KUKA KRL program: EPS_2_251825_SA33_A_20260116064116.src

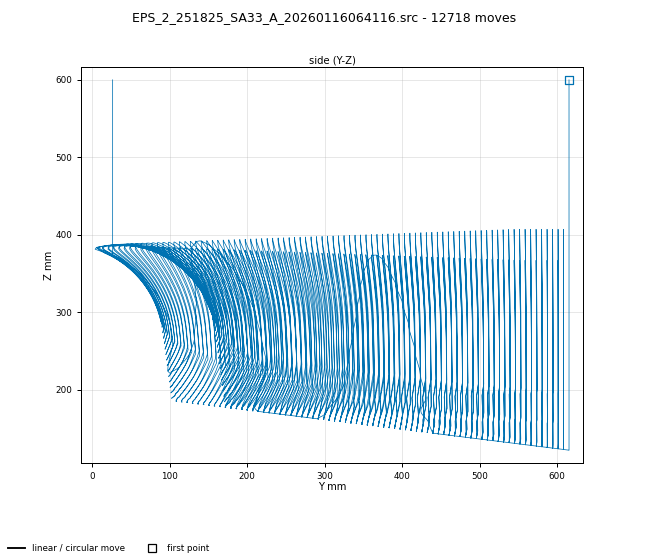
[picture p0: tool path of EPS_2_251825_SA33_A_20260116064116.src, 12718 of 12720 moves have a stored position in this frame; points joined in program order, loops and branches not executed]
&ACCESS RVP
&REL 4
&COMMENT QRS 19112012
&PARAM EDITMASK = *
DEF PART()
EXT BAS (BAS_COMMAND :IN,REAL :IN )
INT I
BAS (#INITMOV,0 )

;KUKA QRS Post kuka4.cps  Date:22-06-2017 !

File_ID=2980

QRS_PRE_INIT()

;Init var - Until changes are made in qrs_pre_init
Outlet_Square_prg=0
Inlet_1_Square_prg=0
Inlet_2_Square_prg=0
Inlet_3_Square_prg=0
Inlet_4_Square_prg=0
Inlet_5_Square_prg=0

Outlet_1={X 0.000, Y 546.330, Z 306.500, B 0.000, E1 0.000 }
Inlet_1={X 0.000, Y 549.180, Z 266.500, B 0.000, E1 202.000 }
Outlet_1_type=201
Inlet_1_type=201
;QRS#1=Sidecore dimensions
;QRS#2=200-8" PVC SDR 35
;QRS#3=200-8" PVC SDR 35
;QRS#4=
;QRS#5=
;QRS#6=
;QRS#7=
;QRS#8=
;QRS#9=12-08 PSX
;QRS#10=12-08 PSX
;QRS#11=
;QRS#12=
;QRS#13=
;QRS#14=
;QRS#15=
;QRS#16=1220x127x686 2,25'
;QRS#17=EPS Height
;QRS#18=407
;QRS#19=*
;QRS#20= UPDATED VERSION 22-06-2017
;QRS#21=*
Outlet_Square=0100
Inlet_1_Square=0100
Inlet_2_Square=0
Inlet_3_Square=0
Inlet_4_Square=0
Inlet_5_Square=0
Mill_Square=1
Outlet_Square_Prg=204
Inlet_1_Square_prg=204

QRS_INIT()

$ADVANCE=5

; T1
PTP {E1 173.647,E2 173.647}
PTP {X 0,Y 615.463,A -85,B 0,C 180,E1 173.647,E2 173.647,E3 0,E4 0,E5 0,E6 0}
QRS_SPEED_INIT()
LIN {X 0,Y 615.463,Z 600,A -85,B 0,C 180,E1 173.647,E2 173.647,E3 0,E4 0,E5 0,E6 0} C_VEL
LIN {X 0,Y 615.463,Z 131.877,A -85,B 0,C 180,E1 173.647,E2 173.647} C_VEL
LIN {X 0,Y 615.463,Z 123.698,A -85,B 0,C 180,E1 173.647,E2 173.647} C_VEL
LIN {X 0,Y 615.445,Z 121.698,A -85,B 0,C 180,E1 173.461,E2 173.461} C_VEL
LIN {X 0,Y 615.439,Z 121.698,A -85,B 0,C 180,E1 171.463,E2 171.463} C_VEL
LIN {X 0,Y 615.428,Z 121.696,A -85,B 0,C 180,E1 169.143,E2 169.143} C_VEL
LIN {X 0,Y 615.442,Z 121.695,A -85,B 0,C 180,E1 166.798,E2 166.798} C_VEL
LIN {X 0,Y 615.481,Z 121.702,A -85,B 0,C 180,E1 164.095,E2 164.095} C_VEL
LIN {X 0,Y 615.427,Z 121.697,A -85,B 0,C 180,E1 161.353,E2 161.353} C_VEL
LIN {X 0,Y 615.486,Z 121.694,A -85,B 0,C 180,E1 158.569,E2 158.569} C_VEL
LIN {X 0,Y 615.433,Z 121.698,A -85,B 0,C 180,E1 155.726,E2 155.726} C_VEL
LIN {X 0,Y 615.425,Z 121.697,A -85,B 0,C 180,E1 153.554,E2 153.554} C_VEL
LIN {X 0,Y 615.493,Z 121.698,A -85,B 0,C 180,E1 150.595,E2 150.595} C_VEL
LIN {X 0,Y 615.468,Z 121.699,A -85,B 0,C 180,E1 148.314,E2 148.314} C_VEL
LIN {X 0,Y 615.433,Z 121.698,A -85,B 0,C 180,E1 145.975,E2 145.975} C_VEL
LIN {X 0,Y 615.427,Z 121.697,A -85,B 0,C 180,E1 143.572,E2 143.572} C_VEL
LIN {X 0,Y 615.49,Z 121.695,A -85,B 0,C 180,E1 140.938,E2 140.938} C_VEL
LIN {X 0,Y 615.465,Z 121.699,A -85,B 0,C 180,E1 138.525,E2 138.525} C_VEL
LIN {X 0,Y 615.424,Z 121.698,A -85,B 0,C 180,E1 136.009,E2 136.009} C_VEL
LIN {X 0,Y 615.423,Z 121.698,A -85,B 0,C 180,E1 133.992,E2 133.992} C_VEL
LIN {X 0,Y 615.448,Z 121.696,A -85,B 0,C 180,E1 131.478,E2 131.478} C_VEL
LIN {X 0,Y 615.485,Z 121.7,A -85,B 0,C 180,E1 128.905,E2 128.905} C_VEL
LIN {X 0,Y 615.43,Z 121.698,A -85,B 0,C 180,E1 126.429,E2 126.429} C_VEL
LIN {X 0,Y 615.422,Z 121.698,A -85,B 0,C 180,E1 124.026,E2 124.026} C_VEL
LIN {X 0,Y 615.445,Z 121.697,A -85,B 0,C 180,E1 121.688,E2 121.688} C_VEL
LIN {X 0,Y 615.479,Z 121.698,A -85,B 0,C 180,E1 119.407,E2 119.407} C_VEL
LIN {X 0,Y 615.421,Z 121.698,A -85,B 0,C 180,E1 116.448,E2 116.448} C_VEL
LIN {X 0,Y 615.436,Z 121.697,A -85,B 0,C 180,E1 113.999,E2 113.999} C_VEL
LIN {X 0,Y 615.498,Z 121.7,A -85,B 0,C 180,E1 111.432,E2 111.432} C_VEL
LIN {X 0,Y 615.419,Z 121.698,A -85,B 0,C 180,E1 108.588,E2 108.588} C_VEL
LIN {X 0,Y 615.462,Z 121.697,A -85,B 0,C 180,E1 105.906,E2 105.906} C_VEL
LIN {X 0,Y 615.444,Z 121.699,A -85,B 0,C 180,E1 103.202,E2 103.202} C_VEL
LIN {X 0,Y 615.417,Z 121.699,A -85,B 0,C 180,E1 100.858,E2 100.858} C_VEL
LIN {X 0,Y 615.423,Z 121.698,A -85,B 0,C 180,E1 98.538,E2 98.538} C_VEL
LIN {X 0,Y 615.496,Z 121.697,A -85,B 0,C 180,E1 95.899,E2 95.899} C_VEL
LIN {X 0,Y 615.429,Z 121.699,A -85,B 0,C 180,E1 93.273,E2 93.273} C_VEL
LIN {X 0,Y 615.429,Z 121.699,A -85,B 0,C 180,E1 91.309,E2 91.309} C_VEL
LIN {X 0,Y 615.427,Z 121.699,A -85,B 0,C 180,E1 89.346,E2 89.346} C_VEL
LIN {X 0,Y 615.427,Z 121.699,A -85,B 0,C 180,E1 87.382,E2 87.382} C_VEL
LIN {X 0,Y 615.434,Z 121.811,A -85,B 0,C 180,E1 86.604,E2 86.604} C_VEL
LIN {X 0,Y 615.454,Z 138.456,A -85,B 0,C 180,E1 83.781,E2 83.781} C_VEL
LIN {X 0,Y 615.439,Z 154.279,A -85,B 0,C 180,E1 81.132,E2 81.132} C_VEL
LIN {X 0,Y 615.46,Z 156.135,A -85,B 0,C 180,E1 80.822,E2 80.822} C_VEL
LIN {X 0,Y 615.446,Z 263.403,A -85,B 0,C 180,E1 79.535,E2 79.535} C_VEL
LIN {X 0,Y 615.449,Z 276.074,A -85,B 0,C 180,E1 79.254,E2 79.254} C_VEL
LIN {X 0,Y 615.477,Z 288.507,A -85,B 0,C 180,E1 78.846,E2 78.846} C_VEL
LIN {X 0,Y 615.497,Z 300.645,A -85,B 0,C 180,E1 78.307,E2 78.307} C_VEL
LIN {X 0,Y 615.483,Z 312.21,A -85,B 0,C 180,E1 77.637,E2 77.637} C_VEL
LIN {X 0,Y 615.498,Z 322.624,A -85,B 0,C 180,E1 76.883,E2 76.883} C_VEL
LIN {X 0,Y 615.497,Z 331.842,A -85,B 0,C 180,E1 76.06,E2 76.06} C_VEL
LIN {X 0,Y 615.496,Z 340.437,A -85,B 0,C 180,E1 75.113,E2 75.113} C_VEL
LIN {X 0,Y 615.497,Z 347.906,A -85,B 0,C 180,E1 74.095,E2 74.095} C_VEL
LIN {X 0,Y 615.496,Z 353.873,A -85,B 0,C 180,E1 73.072,E2 73.072} C_VEL
LIN {X 0,Y 615.498,Z 358.543,A -85,B 0,C 180,E1 72.043,E2 72.043} C_VEL
LIN {X 0,Y 615.494,Z 362.068,A -85,B 0,C 180,E1 71.009,E2 71.009} C_VEL
LIN {X 0,Y 615.495,Z 364.527,A -85,B 0,C 180,E1 69.967,E2 69.967} C_VEL
LIN {X 0,Y 615.497,Z 365.572,A -85,B 0,C 180,E1 69.27,E2 69.27} C_VEL
LIN {X 0,Y 615.498,Z 366.202,A -85,B 0,C 180,E1 68.569,E2 68.569} C_VEL
LIN {X 0,Y 615.497,Z 366.321,A -85,B 0,C 180,E1 67.65,E2 67.65} C_VEL
LIN {X 0,Y 615.496,Z 365.342,A -85,B 0,C 180,E1 66.444,E2 66.444} C_VEL
LIN {X 0,Y 615.494,Z 364.093,A -85,B 0,C 180,E1 65.728,E2 65.728} C_VEL
LIN {X 0,Y 615.495,Z 362.354,A -85,B 0,C 180,E1 65.009,E2 65.009} C_VEL
LIN {X 0,Y 615.496,Z 358.747,A -85,B 0,C 180,E1 63.921,E2 63.921} C_VEL
LIN {X 0,Y 615.494,Z 353.798,A -85,B 0,C 180,E1 62.823,E2 62.823} C_VEL
LIN {X 0,Y 615.496,Z 347.915,A -85,B 0,C 180,E1 61.816,E2 61.816} C_VEL
LIN {X 0,Y 615.496,Z 340.312,A -85,B 0,C 180,E1 60.782,E2 60.782} C_VEL
LIN {X 0,Y 615.496,Z 331.75,A -85,B 0,C 180,E1 59.84,E2 59.84} C_VEL
LIN {X 0,Y 615.497,Z 322.228,A -85,B 0,C 180,E1 58.996,E2 58.996} C_VEL
LIN {X 0,Y 615.471,Z 311.616,A -85,B 0,C 180,E1 58.234,E2 58.234} C_VEL
LIN {X 0,Y 615.467,Z 300.715,A -85,B 0,C 180,E1 57.606,E2 57.606} C_VEL
LIN {X 0,Y 615.494,Z 288.315,A -85,B 0,C 180,E1 57.057,E2 57.057} C_VEL
LIN {X 0,Y 615.49,Z 275.924,A -85,B 0,C 180,E1 56.653,E2 56.653} C_VEL
LIN {X 0,Y 615.467,Z 263.343,A -85,B 0,C 180,E1 56.375,E2 56.375} C_VEL
LIN {X 0,Y 615.49,Z 156.109,A -85,B 0,C 180,E1 55.085,E2 55.085} C_VEL
LIN {X 0,Y 615.471,Z 139.904,A -85,B 0,C 180,E1 52.373,E2 52.373} C_VEL
LIN {X 0,Y 615.484,Z 123.817,A -85,B 0,C 180,E1 49.651,E2 49.651} C_VEL
LIN {X 0,Y 615.48,Z 121.688,A -85,B 0,C 180,E1 49.271,E2 49.271} C_VEL
LIN {X 0,Y 615.486,Z 121.684,A -85,B 0,C 180,E1 46.755,E2 46.755} C_VEL
LIN {X 0,Y 615.488,Z 121.7,A -85,B 0,C 180,E1 43.997,E2 43.997} C_VEL
LIN {X 0,Y 615.487,Z 121.683,A -85,B 0,C 180,E1 41.094,E2 41.094} C_VEL
LIN {X 0,Y 615.487,Z 121.686,A -85,B 0,C 180,E1 38.903,E2 38.903} C_VEL
LIN {X 0,Y 615.487,Z 121.7,A -85,B 0,C 180,E1 36.424,E2 36.424} C_VEL
LIN {X 0,Y 615.478,Z 121.685,A -85,B 0,C 180,E1 33.533,E2 33.533} C_VEL
LIN {X 0,Y 615.484,Z 121.691,A -85,B 0,C 180,E1 30.919,E2 30.919} C_VEL
LIN {X 0,Y 615.484,Z 121.698,A -85,B 0,C 180,E1 28.449,E2 28.449} C_VEL
LIN {X 0,Y 615.483,Z 121.685,A -85,B 0,C 180,E1 25.567,E2 25.567} C_VEL
LIN {X 0,Y 615.49,Z 121.7,A -85,B 0,C 180,E1 22.844,E2 22.844} C_VEL
LIN {X 0,Y 615.472,Z 121.696,A -85,B 0,C 180,E1 20.553,E2 20.553} C_VEL
LIN {X 0,Y 615.468,Z 121.687,A -85,B 0,C 180,E1 17.957,E2 17.957} C_VEL
LIN {X 0,Y 615.493,Z 121.695,A -85,B 0,C 180,E1 15.225,E2 15.225} C_VEL
LIN {X 0,Y 615.457,Z 121.693,A -85,B 0,C 180,E1 12.53,E2 12.53} C_VEL
LIN {X 0,Y 615.491,Z 121.685,A -85,B 0,C 180,E1 9.862,E2 9.862} C_VEL
LIN {X 0,Y 615.48,Z 121.701,A -85,B 0,C 180,E1 7.215,E2 7.215} C_VEL
LIN {X 0,Y 615.451,Z 121.692,A -85,B 0,C 180,E1 4.584,E2 4.584} C_VEL
LIN {X 0,Y 615.5,Z 121.686,A -85,B 0,C 180,E1 1.963,E2 1.963} C_VEL
LIN {X 0,Y 615.472,Z 121.698,A -85,B 0,C 180,E1 -0.655,E2 -0.655} C_VEL
LIN {X 0,Y 615.469,Z 121.698,A -85,B 0,C 180,E1 -2.618,E2 -2.618} C_VEL
LIN {X 0,Y 615.443,Z 121.693,A -85,B 0,C 180,E1 -5.242,E2 -5.242} C_VEL
LIN {X 0,Y 615.489,Z 121.693,A -85,B 0,C 180,E1 -7.876,E2 -7.876} C_VEL
LIN {X 0,Y 615.452,Z 121.697,A -85,B 0,C 180,E1 -10.528,E2 -10.528} C_VEL
LIN {X 0,Y 615.446,Z 121.697,A -85,B 0,C 180,E1 -12.531,E2 -12.531} C_VEL
LIN {X 0,Y 615.437,Z 121.698,A -85,B 0,C 180,E1 -14.551,E2 -14.551} C_VEL
LIN {X 0,Y 615.435,Z 121.697,A -85,B 0,C 180,E1 -16.589,E2 -16.589} C_VEL
LIN {X 0,Y 615.431,Z 121.696,A -85,B 0,C 180,E1 -18.648,E2 -18.648} C_VEL
LIN {X 0,Y 615.487,Z 121.694,A -85,B 0,C 180,E1 -21.432,E2 -21.432} C_VEL
LIN {X 0,Y 615.432,Z 121.698,A -85,B 0,C 180,E1 -24.275,E2 -24.275} C_VEL
LIN {X 0,Y 615.42,Z 121.699,A -85,B 0,C 180,E1 -26.448,E2 -26.448} C_VEL
LIN {X 0,Y 615.491,Z 121.701,A -85,B 0,C 180,E1 -29.407,E2 -29.407} C_VEL
LIN {X 0,Y 615.455,Z 121.7,A -85,B 0,C 180,E1 -31.688,E2 -31.688} C_VEL
LIN {X 0,Y 615.421,Z 121.7,A -85,B 0,C 180,E1 -34.027,E2 -34.027} C_VEL
LIN {X 0,Y 615.463,Z 121.7,A -85,B 0,C 180,E1 -36.933,E2 -36.933} C_VEL
LIN {X 0,Y 615.422,Z 121.7,A -85,B 0,C 180,E1 -39.756,E2 -39.756} C_VEL
LIN {X 0,Y 615.416,Z 121.699,A -85,B 0,C 180,E1 -42.073,E2 -42.073} C_VEL
LIN {X 0,Y 615.421,Z 121.699,A -85,B 0,C 180,E1 -44.156,E2 -44.156} C_VEL
LIN {X 0,Y 615.484,Z 121.7,A -85,B 0,C 180,E1 -46.755,E2 -46.755} C_VEL
LIN {X 0,Y 615.441,Z 121.697,A -85,B 0,C 180,E1 -49.39,E2 -49.39} C_VEL
LIN {X 0,Y 615.428,Z 121.698,A -85,B 0,C 180,E1 -51.927,E2 -51.927} C_VEL
LIN {X 0,Y 615.47,Z 121.699,A -85,B 0,C 180,E1 -54.383,E2 -54.383} C_VEL
LIN {X 0,Y 615.486,Z 121.695,A -85,B 0,C 180,E1 -56.764,E2 -56.764} C_VEL
LIN {X 0,Y 615.453,Z 121.693,A -85,B 0,C 180,E1 -59.078,E2 -59.078} C_VEL
LIN {X 0,Y 615.435,Z 121.696,A -85,B 0,C 180,E1 -61.559,E2 -61.559} C_VEL
LIN {X 0,Y 615.494,Z 121.695,A -85,B 0,C 180,E1 -64.431,E2 -64.431} C_VEL
LIN {X 0,Y 615.442,Z 121.693,A -85,B 0,C 180,E1 -67.154,E2 -67.154} C_VEL
LIN {X 0,Y 615.441,Z 121.788,A -85,B 0,C 180,E1 -67.44,E2 -67.44} C_VEL
LIN {X 0,Y 615.477,Z 140.398,A -85,B 0,C 180,E1 -69.967,E2 -69.967} C_VEL
LIN {X 0,Y 615.47,Z 161.077,A -85,B 0,C 180,E1 -72.729,E2 -72.729} C_VEL
LIN {X 0,Y 615.472,Z 181.733,A -85,B 0,C 180,E1 -75.451,E2 -75.451} C_VEL
LIN {X 0,Y 615.454,Z 194.471,A -85,B 0,C 180,E1 -77.113,E2 -77.113} C_VEL
LIN {X 0,Y 615.488,Z 302.833,A -85,B 0,C 180,E1 -78.411,E2 -78.411} C_VEL
LIN {X 0,Y 615.477,Z 315.348,A -85,B 0,C 180,E1 -78.682,E2 -78.682} C_VEL
LIN {X 0,Y 615.488,Z 328.62,A -85,B 0,C 180,E1 -79.113,E2 -79.113} C_VEL
LIN {X 0,Y 615.477,Z 340.48,A -85,B 0,C 180,E1 -79.639,E2 -79.639} C_VEL
LIN {X 0,Y 615.494,Z 351.995,A -85,B 0,C 180,E1 -80.304,E2 -80.304} C_VEL
LIN {X 0,Y 615.499,Z 362.342,A -85,B 0,C 180,E1 -81.05,E2 -81.05} C_VEL
LIN {X 0,Y 615.497,Z 370.813,A -85,B 0,C 180,E1 -81.794,E2 -81.794} C_VEL
LIN {X 0,Y 615.498,Z 378.607,A -85,B 0,C 180,E1 -82.62,E2 -82.62} C_VEL
LIN {X 0,Y 615.496,Z 386.204,A -85,B 0,C 180,E1 -83.608,E2 -83.608} C_VEL
LIN {X 0,Y 615.498,Z 393.205,A -85,B 0,C 180,E1 -84.759,E2 -84.759} C_VEL
LIN {X 0,Y 615.494,Z 397.852,A -85,B 0,C 180,E1 -85.744,E2 -85.744} C_VEL
LIN {X 0,Y 615.494,Z 401.399,A -85,B 0,C 180,E1 -86.727,E2 -86.727} C_VEL
LIN {X 0,Y 615.497,Z 403.233,A -85,B 0,C 180,E1 -87.382,E2 -87.382} C_VEL
LIN {X 0,Y 615.5,Z 404.608,A -85,B 0,C 180,E1 -88.037,E2 -88.037} C_VEL
LIN {X 0,Y 615.496,Z 406.174,A -85,B 0,C 180,E1 -89.346,E2 -89.346} C_VEL
LIN {X 0,Y 615.494,Z 406.389,A -85,B 0,C 180,E1 -90,E2 -90} C_VEL
LIN {X 0,Y 615.495,Z 405.58,A -85,B 0,C 180,E1 -91.309,E2 -91.309} C_VEL
LIN {X 0,Y 615.5,Z 404.607,A -85,B 0,C 180,E1 -91.963,E2 -91.963} C_VEL
LIN {X 0,Y 615.497,Z 403.233,A -85,B 0,C 180,E1 -92.618,E2 -92.618} C_VEL
LIN {X 0,Y 615.496,Z 400.349,A -85,B 0,C 180,E1 -93.601,E2 -93.601} C_VEL
LIN {X 0,Y 615.498,Z 396.441,A -85,B 0,C 180,E1 -94.585,E2 -94.585} C_VEL
LIN {X 0,Y 615.499,Z 391.404,A -85,B 0,C 180,E1 -95.57,E2 -95.57} C_VEL
LIN {X 0,Y 615.497,Z 384.87,A -85,B 0,C 180,E1 -96.583,E2 -96.583} C_VEL
LIN {X 0,Y 615.497,Z 377.131,A -85,B 0,C 180,E1 -97.546,E2 -97.546} C_VEL
LIN {X 0,Y 615.498,Z 369.043,A -85,B 0,C 180,E1 -98.371,E2 -98.371} C_VEL
LIN {X 0,Y 615.499,Z 359.165,A -85,B 0,C 180,E1 -99.199,E2 -99.199} C_VEL
LIN {X 0,Y 615.488,Z 347.978,A -85,B 0,C 180,E1 -99.945,E2 -99.945} C_VEL
LIN {X 0,Y 615.482,Z 337.019,A -85,B 0,C 180,E1 -100.527,E2 -100.527} C_VEL
LIN {X 0,Y 615.48,Z 324.488,A -85,B 0,C 180,E1 -101.04,E2 -101.04} C_VEL
LIN {X 0,Y 615.479,Z 312.057,A -85,B 0,C 180,E1 -101.402,E2 -101.402} C_VEL
LIN {X 0,Y 615.493,Z 298.449,A -85,B 0,C 180,E1 -101.652,E2 -101.652} C_VEL
LIN {X 0,Y 615.454,Z 194.469,A -85,B 0,C 180,E1 -102.887,E2 -102.887} C_VEL
LIN {X 0,Y 615.496,Z 172.694,A -85,B 0,C 180,E1 -105.735,E2 -105.735} C_VEL
LIN {X 0,Y 615.455,Z 152.319,A -85,B 0,C 180,E1 -108.436,E2 -108.436} C_VEL
LIN {X 0,Y 615.475,Z 132.635,A -85,B 0,C 180,E1 -111.082,E2 -111.082} C_VEL
LIN {X 0,Y 615.44,Z 121.695,A -85,B 0,C 180,E1 -112.592,E2 -112.592} C_VEL
LIN {X 0,Y 615.452,Z 121.692,A -85,B 0,C 180,E1 -114.994,E2 -114.994} C_VEL
LIN {X 0,Y 615.475,Z 121.699,A -85,B 0,C 180,E1 -117.916,E2 -117.916} C_VEL
LIN {X 0,Y 615.449,Z 121.697,A -85,B 0,C 180,E1 -120.163,E2 -120.163} C_VEL
LIN {X 0,Y 615.438,Z 121.694,A -85,B 0,C 180,E1 -122.461,E2 -122.461} C_VEL
LIN {X 0,Y 615.454,Z 121.692,A -85,B 0,C 180,E1 -124.818,E2 -124.818} C_VEL
LIN {X 0,Y 615.497,Z 121.692,A -85,B 0,C 180,E1 -127.242,E2 -127.242} C_VEL
LIN {X 0,Y 615.462,Z 121.698,A -85,B 0,C 180,E1 -129.753,E2 -129.753} C_VEL
LIN {X 0,Y 615.439,Z 121.694,A -85,B 0,C 180,E1 -132.358,E2 -132.358} C_VEL
LIN {X 0,Y 615.497,Z 121.692,A -85,B 0,C 180,E1 -135.068,E2 -135.068} C_VEL
LIN {X 0,Y 615.454,Z 121.698,A -85,B 0,C 180,E1 -137.644,E2 -137.644} C_VEL
LIN {X 0,Y 615.438,Z 121.694,A -85,B 0,C 180,E1 -140.246,E2 -140.246} C_VEL
LIN {X 0,Y 615.488,Z 121.701,A -85,B 0,C 180,E1 -143.064,E2 -143.064} C_VEL
LIN {X 0,Y 615.435,Z 121.695,A -85,B 0,C 180,E1 -145.974,E2 -145.974} C_VEL
LIN {X 0,Y 615.485,Z 121.701,A -85,B 0,C 180,E1 -148.915,E2 -148.915} C_VEL
LIN {X 0,Y 615.438,Z 121.696,A -85,B 0,C 180,E1 -151.559,E2 -151.559} C_VEL
LIN {X 0,Y 615.437,Z 121.696,A -85,B 0,C 180,E1 -153.553,E2 -153.553} C_VEL
LIN {X 0,Y 615.444,Z 121.694,A -85,B 0,C 180,E1 -156.002,E2 -156.002} C_VEL
LIN {X 0,Y 615.498,Z 121.694,A -85,B 0,C 180,E1 -158.568,E2 -158.568} C_VEL
LIN {X 0,Y 615.434,Z 121.696,A -85,B 0,C 180,E1 -161.412,E2 -161.412} C_VEL
LIN {X 0,Y 615.433,Z 121.695,A -85,B 0,C 180,E1 -163.588,E2 -163.588} C_VEL
LIN {X 0,Y 615.475,Z 121.692,A -85,B 0,C 180,E1 -166.125,E2 -166.125} C_VEL
LIN {X 0,Y 615.46,Z 121.699,A -85,B 0,C 180,E1 -168.806,E2 -168.806} C_VEL
LIN {X 0,Y 615.456,Z 121.698,A -85,B 0,C 180,E1 -170.8,E2 -170.8} C_VEL
LIN {X 0,Y 615.453,Z 121.698,A -85,B 0,C 180,E1 -172.783,E2 -172.783} C_VEL
LIN {X 0,Y 615.451,Z 121.698,A -85,B 0,C 180,E1 -174.758,E2 -174.758} C_VEL
LIN {X 0,Y 615.45,Z 121.698,A -85,B 0,C 180,E1 -176.726,E2 -176.726} C_VEL
LIN {X 0,Y 615.449,Z 121.698,A -85,B 0,C 180,E1 -178.691,E2 -178.691} C_VEL
LIN {X 0,Y 615.447,Z 121.698,A -85,B 0,C 180,E1 -180.654,E2 -180.654} C_VEL
LIN {X 0,Y 615.447,Z 121.698,A -85,B 0,C 180,E1 -182.617,E2 -182.617} C_VEL
LIN {X 0,Y 615.445,Z 121.698,A -85,B 0,C 180,E1 -184.584,E2 -184.584} C_VEL
LIN {X 0,Y 615.445,Z 121.698,A -85,B 0,C 180,E1 -186.539,E2 -186.539} C_VEL
LIN {X 0,Y 614.76,Z 121.842,A -85,B 0,C 180,E1 -187.085,E2 -187.085} C_VEL
LIN {X 0,Y 611.917,Z 122.266,A -85,B 0,C 180,E1 -187.972,E2 -187.972} C_VEL
LIN {X 0,Y 609.532,Z 122.568,A -85,B 0,C 180,E1 -188.684,E2 -188.684} C_VEL
LIN {X 0,Y 608.513,Z 122.682,A -85,B 0,C 180,E1 -189.234,E2 -189.234} C_VEL
LIN {X 0,Y 608.432,Z 122.692,A -85,B 0,C 180,E1 -189.42,E2 -189.42} C_VEL
LIN {X 0,Y 608.455,Z 122.697,A -85,B 0,C 180,E1 -191.999,E2 -191.999} C_VEL
LIN {X 0,Y 608.4,Z 122.694,A -85,B 0,C 180,E1 -194.722,E2 -194.722} C_VEL
LIN {X 0,Y 608.411,Z 122.693,A -85,B 0,C 180,E1 -196.785,E2 -196.785} C_VEL
LIN {X 0,Y 608.434,Z 122.697,A -85,B 0,C 180,E1 -199.571,E2 -199.571} C_VEL
LIN {X 0,Y 608.416,Z 122.693,A -85,B 0,C 180,E1 -202.407,E2 -202.407} C_VEL
LIN {X 0,Y 608.414,Z 122.692,A -85,B 0,C 180,E1 -204.572,E2 -204.572} C_VEL
LIN {X 0,Y 608.461,Z 122.691,A -85,B 0,C 180,E1 -207.203,E2 -207.203} C_VEL
LIN {X 0,Y 608.419,Z 122.695,A -85,B 0,C 180,E1 -209.963,E2 -209.963} C_VEL
LIN {X 0,Y 608.412,Z 122.693,A -85,B 0,C 180,E1 -212.514,E2 -212.514} C_VEL
LIN {X 0,Y 608.416,Z 122.695,A -85,B 0,C 180,E1 -214.9,E2 -214.9} C_VEL
LIN {X 0,Y 608.436,Z 122.693,A -85,B 0,C 180,E1 -217.748,E2 -217.748} C_VEL
LIN {X 0,Y 608.399,Z 122.694,A -85,B 0,C 180,E1 -220.323,E2 -220.323} C_VEL
LIN {X 0,Y 608.444,Z 122.695,A -85,B 0,C 180,E1 -222.96,E2 -222.96} C_VEL
LIN {X 0,Y 608.409,Z 122.695,A -85,B 0,C 180,E1 -225.74,E2 -225.74} C_VEL
LIN {X 0,Y 608.408,Z 122.693,A -85,B 0,C 180,E1 -227.934,E2 -227.934} C_VEL
LIN {X 0,Y 608.435,Z 122.695,A -85,B 0,C 180,E1 -230.705,E2 -230.705} C_VEL
LIN {X 0,Y 608.45,Z 122.696,A -85,B 0,C 180,E1 -233.084,E2 -233.084} C_VEL
LIN {X 0,Y 608.425,Z 122.692,A -85,B 0,C 180,E1 -235.527,E2 -235.527} C_VEL
LIN {X 0,Y 608.415,Z 122.692,A -85,B 0,C 180,E1 -237.902,E2 -237.902} C_VEL
LIN {X 0,Y 608.428,Z 122.693,A -85,B 0,C 180,E1 -240.218,E2 -240.218} C_VEL
LIN {X 0,Y 608.467,Z 122.695,A -85,B 0,C 180,E1 -242.793,E2 -242.793} C_VEL
LIN {X 0,Y 608.409,Z 122.693,A -85,B 0,C 180,E1 -245.427,E2 -245.427} C_VEL
LIN {X 0,Y 608.454,Z 122.693,A -85,B 0,C 180,E1 -248.308,E2 -248.308} C_VEL
LIN {X 0,Y 608.406,Z 122.694,A -85,B 0,C 180,E1 -251.3,E2 -251.3} C_VEL
LIN {X 0,Y 608.423,Z 122.693,A -85,B 0,C 180,E1 -253.905,E2 -253.905} C_VEL
LIN {X 0,Y 608.43,Z 122.696,A -85,B 0,C 180,E1 -256.643,E2 -256.643} C_VEL
LIN {X 0,Y 608.4,Z 122.694,A -85,B 0,C 180,E1 -259.349,E2 -259.349} C_VEL
LIN {X 0,Y 608.463,Z 122.693,A -85,B 0,C 180,E1 -262.033,E2 -262.033} C_VEL
LIN {X 0,Y 608.419,Z 122.694,A -85,B 0,C 180,E1 -264.698,E2 -264.698} C_VEL
LIN {X 0,Y 608.42,Z 122.692,A -85,B 0,C 180,E1 -267.352,E2 -267.352} C_VEL
LIN {X 0,Y 608.469,Z 122.695,A -85,B 0,C 180,E1 -270,E2 -270} C_VEL
LIN {X 0,Y 608.422,Z 122.693,A -85,B 0,C 180,E1 -272.648,E2 -272.648} C_VEL
LIN {X 0,Y 608.414,Z 122.794,A -85,B 0,C 180,E1 -273.332,E2 -273.332} C_VEL
LIN {X 0,Y 608.461,Z 139.275,A -85,B 0,C 180,E1 -276.152,E2 -276.152} C_VEL
LIN {X 0,Y 608.415,Z 154.004,A -85,B 0,C 180,E1 -278.637,E2 -278.637} C_VEL
LIN {X 0,Y 608.426,Z 156.373,A -85,B 0,C 180,E1 -279.034,E2 -279.034} C_VEL
LIN {X 0,Y 608.503,Z 263.641,A -85,B 0,C 180,E1 -280.334,E2 -280.334} C_VEL
LIN {X 0,Y 608.494,Z 277.407,A -85,B 0,C 180,E1 -280.649,E2 -280.649} C_VEL
LIN {X 0,Y 608.511,Z 289.332,A -85,B 0,C 180,E1 -281.054,E2 -281.054} C_VEL
LIN {X 0,Y 608.505,Z 300.864,A -85,B 0,C 180,E1 -281.576,E2 -281.576} C_VEL
LIN {X 0,Y 608.488,Z 312.454,A -85,B 0,C 180,E1 -282.253,E2 -282.253} C_VEL
LIN {X 0,Y 608.496,Z 322.908,A -85,B 0,C 180,E1 -283.016,E2 -283.016} C_VEL
LIN {X 0,Y 608.456,Z 332.698,A -85,B 0,C 180,E1 -283.901,E2 -283.901} C_VEL
LIN {X 0,Y 608.451,Z 341.527,A -85,B 0,C 180,E1 -284.892,E2 -284.892} C_VEL
LIN {X 0,Y 608.461,Z 348.912,A -85,B 0,C 180,E1 -285.922,E2 -285.922} C_VEL
LIN {X 0,Y 608.454,Z 355.63,A -85,B 0,C 180,E1 -287.13,E2 -287.13} C_VEL
LIN {X 0,Y 608.43,Z 360.054,A -85,B 0,C 180,E1 -288.172,E2 -288.172} C_VEL
LIN {X 0,Y 608.429,Z 362.389,A -85,B 0,C 180,E1 -288.87,E2 -288.87} C_VEL
LIN {X 0,Y 608.418,Z 364.202,A -85,B 0,C 180,E1 -289.572,E2 -289.572} C_VEL
LIN {X 0,Y 608.439,Z 366.128,A -85,B 0,C 180,E1 -290.674,E2 -290.674} C_VEL
LIN {X 0,Y 608.418,Z 366.924,A -85,B 0,C 180,E1 -291.693,E2 -291.693} C_VEL
LIN {X 0,Y 608.421,Z 366.906,A -85,B 0,C 180,E1 -292.47,E2 -292.47} C_VEL
LIN {X 0,Y 608.43,Z 366.47,A -85,B 0,C 180,E1 -293.125,E2 -293.125} C_VEL
LIN {X 0,Y 608.424,Z 365.007,A -85,B 0,C 180,E1 -294.143,E2 -294.143} C_VEL
LIN {X 0,Y 608.439,Z 362.129,A -85,B 0,C 180,E1 -295.302,E2 -295.302} C_VEL
LIN {X 0,Y 608.453,Z 358.143,A -85,B 0,C 180,E1 -296.404,E2 -296.404} C_VEL
LIN {X 0,Y 608.439,Z 352.745,A -85,B 0,C 180,E1 -297.519,E2 -297.519} C_VEL
LIN {X 0,Y 608.456,Z 345.893,A -85,B 0,C 180,E1 -298.619,E2 -298.619} C_VEL
LIN {X 0,Y 608.461,Z 338.268,A -85,B 0,C 180,E1 -299.589,E2 -299.589} C_VEL
LIN {X 0,Y 608.474,Z 329.005,A -85,B 0,C 180,E1 -300.545,E2 -300.545} C_VEL
LIN {X 0,Y 608.479,Z 319.853,A -85,B 0,C 180,E1 -301.316,E2 -301.316} C_VEL
LIN {X 0,Y 608.475,Z 310.005,A -85,B 0,C 180,E1 -301.996,E2 -301.996} C_VEL
LIN {X 0,Y 608.496,Z 298.187,A -85,B 0,C 180,E1 -302.645,E2 -302.645} C_VEL
LIN {X 0,Y 608.517,Z 285.724,A -85,B 0,C 180,E1 -303.172,E2 -303.172} C_VEL
LIN {X 0,Y 608.52,Z 272.657,A -85,B 0,C 180,E1 -303.568,E2 -303.568} C_VEL
LIN {X 0,Y 608.525,Z 260.478,A -85,B 0,C 180,E1 -303.806,E2 -303.806} C_VEL
LIN {X 0,Y 608.471,Z 156.466,A -85,B 0,C 180,E1 -305.046,E2 -305.046} C_VEL
LIN {X 0,Y 608.466,Z 140.404,A -85,B 0,C 180,E1 -307.747,E2 -307.747} C_VEL
LIN {X 0,Y 608.485,Z 125.247,A -85,B 0,C 180,E1 -310.334,E2 -310.334} C_VEL
LIN {X 0,Y 608.457,Z 122.689,A -85,B 0,C 180,E1 -310.793,E2 -310.793} C_VEL
LIN {X 0,Y 608.474,Z 122.686,A -85,B 0,C 180,E1 -313.31,E2 -313.31} C_VEL
LIN {X 0,Y 608.471,Z 122.692,A -85,B 0,C 180,E1 -316.132,E2 -316.132} C_VEL
LIN {X 0,Y 608.455,Z 122.688,A -85,B 0,C 180,E1 -318.824,E2 -318.824} C_VEL
LIN {X 0,Y 608.468,Z 122.691,A -85,B 0,C 180,E1 -321.413,E2 -321.413} C_VEL
LIN {X 0,Y 608.442,Z 122.694,A -85,B 0,C 180,E1 -323.955,E2 -323.955} C_VEL
LIN {X 0,Y 608.444,Z 122.689,A -85,B 0,C 180,E1 -326.329,E2 -326.329} C_VEL
LIN {X 0,Y 608.446,Z 122.689,A -85,B 0,C 180,E1 -328.733,E2 -328.733} C_VEL
LIN {X 0,Y 608.473,Z 122.695,A -85,B 0,C 180,E1 -331.381,E2 -331.381} C_VEL
LIN {X 0,Y 608.436,Z 122.691,A -85,B 0,C 180,E1 -333.965,E2 -333.965} C_VEL
LIN {X 0,Y 608.452,Z 122.692,A -85,B 0,C 180,E1 -336.877,E2 -336.877} C_VEL
LIN {X 0,Y 608.459,Z 122.694,A -85,B 0,C 180,E1 -339.324,E2 -339.324} C_VEL
LIN {X 0,Y 608.432,Z 122.691,A -85,B 0,C 180,E1 -341.828,E2 -341.828} C_VEL
LIN {X 0,Y 608.473,Z 122.69,A -85,B 0,C 180,E1 -344.595,E2 -344.595} C_VEL
LIN {X 0,Y 608.456,Z 122.69,A -85,B 0,C 180,E1 -347.323,E2 -347.323} C_VEL
LIN {X 0,Y 608.454,Z 122.688,A -85,B 0,C 180,E1 -350.023,E2 -350.023} C_VEL
LIN {X 0,Y 608.461,Z 122.697,A -85,B 0,C 180,E1 -352.701,E2 -352.701} C_VEL
LIN {X 0,Y 608.464,Z 122.695,A -85,B 0,C 180,E1 -354.699,E2 -354.699} C_VEL
LIN {X 0,Y 608.443,Z 122.689,A -85,B 0,C 180,E1 -357.352,E2 -357.352} C_VEL
LIN {X 0,Y 608.477,Z 122.688,A -85,B 0,C 180,E1 -360.001,E2 -360.001} C_VEL
LIN {X 0,Y 608.461,Z 122.692,A -85,B 0,C 180,E1 -362.649,E2 -362.649} C_VEL
LIN {X 0,Y 608.43,Z 122.69,A -85,B 0,C 180,E1 -365.303,E2 -365.303} C_VEL
LIN {X 0,Y 608.477,Z 122.691,A -85,B 0,C 180,E1 -367.967,E2 -367.967} C_VEL
LIN {X 0,Y 608.427,Z 122.693,A -85,B 0,C 180,E1 -370.651,E2 -370.651} C_VEL
LIN {X 0,Y 608.438,Z 122.691,A -85,B 0,C 180,E1 -373.357,E2 -373.357} C_VEL
LIN {X 0,Y 608.446,Z 122.695,A -85,B 0,C 180,E1 -376.095,E2 -376.095} C_VEL
LIN {X 0,Y 608.431,Z 122.69,A -85,B 0,C 180,E1 -378.871,E2 -378.871} C_VEL
LIN {X 0,Y 608.455,Z 122.698,A -85,B 0,C 180,E1 -381.693,E2 -381.693} C_VEL
LIN {X 0,Y 608.413,Z 122.693,A -85,B 0,C 180,E1 -384.573,E2 -384.573} C_VEL
LIN {X 0,Y 608.46,Z 122.692,A -85,B 0,C 180,E1 -387.203,E2 -387.203} C_VEL
LIN {X 0,Y 608.411,Z 122.695,A -85,B 0,C 180,E1 -389.962,E2 -389.962} C_VEL
LIN {X 0,Y 608.407,Z 122.694,A -85,B 0,C 180,E1 -392.514,E2 -392.514} C_VEL
LIN {X 0,Y 608.41,Z 122.697,A -85,B 0,C 180,E1 -394.9,E2 -394.9} C_VEL
LIN {X 0,Y 608.404,Z 122.695,A -85,B 0,C 180,E1 -397.751,E2 -397.751} C_VEL
LIN {X 0,Y 608.404,Z 122.694,A -85,B 0,C 180,E1 -400.324,E2 -400.324} C_VEL
LIN {X 0,Y 608.442,Z 122.699,A -85,B 0,C 180,E1 -402.961,E2 -402.961} C_VEL
LIN {X 0,Y 608.404,Z 122.694,A -85,B 0,C 180,E1 -405.742,E2 -405.742} C_VEL
LIN {X 0,Y 608.407,Z 122.694,A -85,B 0,C 180,E1 -407.934,E2 -407.934} C_VEL
LIN {X 0,Y 608.436,Z 122.7,A -85,B 0,C 180,E1 -410.707,E2 -410.707} C_VEL
LIN {X 0,Y 608.435,Z 122.693,A -85,B 0,C 180,E1 -413.084,E2 -413.084} C_VEL
LIN {X 0,Y 608.429,Z 122.691,A -85,B 0,C 180,E1 -415.528,E2 -415.528} C_VEL
LIN {X 0,Y 608.431,Z 122.692,A -85,B 0,C 180,E1 -417.903,E2 -417.903} C_VEL
LIN {X 0,Y 608.457,Z 122.694,A -85,B 0,C 180,E1 -420.22,E2 -420.22} C_VEL
LIN {X 0,Y 608.409,Z 122.693,A -85,B 0,C 180,E1 -423.224,E2 -423.224} C_VEL
LIN {X 0,Y 608.423,Z 122.692,A -85,B 0,C 180,E1 -425.428,E2 -425.428} C_VEL
LIN {X 0,Y 608.435,Z 122.82,A -85,B 0,C 180,E1 -427.309,E2 -427.309} C_VEL
LIN {X 0,Y 608.573,Z 138.081,A -85,B 0,C 180,E1 -429.413,E2 -429.413} C_VEL
LIN {X 0,Y 608.533,Z 158.53,A -85,B 0,C 180,E1 -432.179,E2 -432.179} C_VEL
LIN {X 0,Y 608.493,Z 179.241,A -85,B 0,C 180,E1 -434.938,E2 -434.938} C_VEL
LIN {X 0,Y 608.441,Z 194.613,A -85,B 0,C 180,E1 -436.962,E2 -436.962} C_VEL
LIN {X 0,Y 608.556,Z 250.597,A -85,B 0,C 180,E1 -437.643,E2 -437.643} C_VEL
LIN {X 0,Y 608.547,Z 302.95,A -85,B 0,C 180,E1 -438.277,E2 -438.277} C_VEL
LIN {X 0,Y 608.512,Z 316.219,A -85,B 0,C 180,E1 -438.572,E2 -438.572} C_VEL
LIN {X 0,Y 608.514,Z 328.631,A -85,B 0,C 180,E1 -438.982,E2 -438.982} C_VEL
LIN {X 0,Y 608.499,Z 340.636,A -85,B 0,C 180,E1 -439.519,E2 -439.519} C_VEL
LIN {X 0,Y 608.484,Z 352.199,A -85,B 0,C 180,E1 -440.191,E2 -440.191} C_VEL
LIN {X 0,Y 608.485,Z 362.595,A -85,B 0,C 180,E1 -440.946,E2 -440.946} C_VEL
LIN {X 0,Y 608.475,Z 371.113,A -85,B 0,C 180,E1 -441.699,E2 -441.699} C_VEL
LIN {X 0,Y 608.471,Z 378.961,A -85,B 0,C 180,E1 -442.534,E2 -442.534} C_VEL
LIN {X 0,Y 608.461,Z 386.288,A -85,B 0,C 180,E1 -443.485,E2 -443.485} C_VEL
LIN {X 0,Y 608.451,Z 391.866,A -85,B 0,C 180,E1 -444.366,E2 -444.366} C_VEL
LIN {X 0,Y 608.432,Z 396.95,A -85,B 0,C 180,E1 -445.362,E2 -445.362} C_VEL
LIN {X 0,Y 608.449,Z 400.897,A -85,B 0,C 180,E1 -446.358,E2 -446.358} C_VEL
LIN {X 0,Y 608.425,Z 403.809,A -85,B 0,C 180,E1 -447.352,E2 -447.352} C_VEL
LIN {X 0,Y 608.445,Z 405.202,A -85,B 0,C 180,E1 -448.014,E2 -448.014} C_VEL
LIN {X 0,Y 608.438,Z 406.784,A -85,B 0,C 180,E1 -449.338,E2 -449.338} C_VEL
LIN {X 0,Y 608.434,Z 407,A -85,B 0,C 180,E1 -450,E2 -450} C_VEL
LIN {X 0,Y 608.448,Z 406.184,A -85,B 0,C 180,E1 -451.324,E2 -451.324} C_VEL
LIN {X 0,Y 608.445,Z 405.201,A -85,B 0,C 180,E1 -451.986,E2 -451.986} C_VEL
LIN {X 0,Y 608.425,Z 403.809,A -85,B 0,C 180,E1 -452.648,E2 -452.648} C_VEL
LIN {X 0,Y 608.449,Z 400.896,A -85,B 0,C 180,E1 -453.643,E2 -453.643} C_VEL
LIN {X 0,Y 608.432,Z 396.949,A -85,B 0,C 180,E1 -454.638,E2 -454.638} C_VEL
LIN {X 0,Y 608.438,Z 390.876,A -85,B 0,C 180,E1 -455.801,E2 -455.801} C_VEL
LIN {X 0,Y 608.462,Z 384.234,A -85,B 0,C 180,E1 -456.799,E2 -456.799} C_VEL
LIN {X 0,Y 608.456,Z 375.987,A -85,B 0,C 180,E1 -457.8,E2 -457.8} C_VEL
LIN {X 0,Y 608.472,Z 367.534,A -85,B 0,C 180,E1 -458.636,E2 -458.636} C_VEL
LIN {X 0,Y 608.479,Z 357.088,A -85,B 0,C 180,E1 -459.474,E2 -459.474} C_VEL
LIN {X 0,Y 608.489,Z 346.753,A -85,B 0,C 180,E1 -460.145,E2 -460.145} C_VEL
LIN {X 0,Y 608.519,Z 335.264,A -85,B 0,C 180,E1 -460.74,E2 -460.74} C_VEL
LIN {X 0,Y 608.528,Z 322.886,A -85,B 0,C 180,E1 -461.225,E2 -461.225} C_VEL
LIN {X 0,Y 608.544,Z 309.429,A -85,B 0,C 180,E1 -461.597,E2 -461.597} C_VEL
LIN {X 0,Y 608.553,Z 297.067,A -85,B 0,C 180,E1 -461.808,E2 -461.808} C_VEL
LIN {X 0,Y 608.496,Z 195.123,A -85,B 0,C 180,E1 -463.016,E2 -463.016} C_VEL
LIN {X 0,Y 608.444,Z 194.126,A -85,B 0,C 180,E1 -463.102,E2 -463.102} C_VEL
LIN {X 0,Y 608.497,Z 172.767,A -85,B 0,C 180,E1 -465.921,E2 -465.921} C_VEL
LIN {X 0,Y 608.499,Z 151.838,A -85,B 0,C 180,E1 -468.723,E2 -468.723} C_VEL
LIN {X 0,Y 608.575,Z 131.344,A -85,B 0,C 180,E1 -471.51,E2 -471.51} C_VEL
LIN {X 0,Y 608.426,Z 122.693,A -85,B 0,C 180,E1 -472.716,E2 -472.716} C_VEL
LIN {X 0,Y 608.438,Z 122.693,A -85,B 0,C 180,E1 -475.302,E2 -475.302} C_VEL
LIN {X 0,Y 608.44,Z 122.696,A -85,B 0,C 180,E1 -477.519,E2 -477.519} C_VEL
LIN {X 0,Y 608.437,Z 122.695,A -85,B 0,C 180,E1 -479.966,E2 -479.966} C_VEL
LIN {X 0,Y 608.423,Z 122.691,A -85,B 0,C 180,E1 -482.516,E2 -482.516} C_VEL
LIN {X 0,Y 608.434,Z 122.696,A -85,B 0,C 180,E1 -485.279,E2 -485.279} C_VEL
LIN {X 0,Y 608.449,Z 122.694,A -85,B 0,C 180,E1 -487.748,E2 -487.748} C_VEL
LIN {X 0,Y 608.409,Z 122.693,A -85,B 0,C 180,E1 -490.324,E2 -490.324} C_VEL
LIN {X 0,Y 608.448,Z 122.692,A -85,B 0,C 180,E1 -492.961,E2 -492.961} C_VEL
LIN {X 0,Y 608.423,Z 122.694,A -85,B 0,C 180,E1 -495.74,E2 -495.74} C_VEL
LIN {X 0,Y 608.423,Z 122.692,A -85,B 0,C 180,E1 -497.935,E2 -497.935} C_VEL
LIN {X 0,Y 608.441,Z 122.692,A -85,B 0,C 180,E1 -500.707,E2 -500.707} C_VEL
LIN {X 0,Y 608.456,Z 122.697,A -85,B 0,C 180,E1 -503.085,E2 -503.085} C_VEL
LIN {X 0,Y 608.445,Z 122.691,A -85,B 0,C 180,E1 -505.529,E2 -505.529} C_VEL
LIN {X 0,Y 608.427,Z 122.691,A -85,B 0,C 180,E1 -507.903,E2 -507.903} C_VEL
LIN {X 0,Y 608.436,Z 122.69,A -85,B 0,C 180,E1 -510.218,E2 -510.218} C_VEL
LIN {X 0,Y 608.485,Z 122.693,A -85,B 0,C 180,E1 -512.793,E2 -512.793} C_VEL
LIN {X 0,Y 608.426,Z 122.692,A -85,B 0,C 180,E1 -515.427,E2 -515.427} C_VEL
LIN {X 0,Y 608.459,Z 122.69,A -85,B 0,C 180,E1 -518.308,E2 -518.308} C_VEL
LIN {X 0,Y 608.421,Z 122.693,A -85,B 0,C 180,E1 -521.3,E2 -521.3} C_VEL
LIN {X 0,Y 608.43,Z 122.691,A -85,B 0,C 180,E1 -523.905,E2 -523.905} C_VEL
LIN {X 0,Y 608.448,Z 122.697,A -85,B 0,C 180,E1 -526.643,E2 -526.643} C_VEL
LIN {X 0,Y 608.416,Z 122.692,A -85,B 0,C 180,E1 -529.349,E2 -529.349} C_VEL
LIN {X 0,Y 608.47,Z 122.689,A -85,B 0,C 180,E1 -532.032,E2 -532.032} C_VEL
LIN {X 0,Y 608.437,Z 122.694,A -85,B 0,C 180,E1 -534.697,E2 -534.697} C_VEL
LIN {X 0,Y 608.431,Z 122.69,A -85,B 0,C 180,E1 -537.351,E2 -537.351} C_VEL
LIN {X 0,Y 608.477,Z 122.691,A -85,B 0,C 180,E1 -539.999,E2 -539.999} C_VEL
LIN {X 0,Y 608.441,Z 122.692,A -85,B 0,C 180,E1 -542.648,E2 -542.648} C_VEL
LIN {X 0,Y 608.421,Z 122.692,A -85,B 0,C 180,E1 -545.302,E2 -545.302} C_VEL
LIN {X 0,Y 608.475,Z 122.694,A -85,B 0,C 180,E1 -547.966,E2 -547.966} C_VEL
LIN {X 0,Y 608.432,Z 122.692,A -85,B 0,C 180,E1 -549.42,E2 -549.42} C_VEL
LIN {X 0,Y 607.775,Z 122.783,A -85,B 0,C 180,E1 -549.973,E2 -549.973} C_VEL
LIN {X 0,Y 604.941,Z 123.137,A -85,B 0,C 180,E1 -550.87,E2 -550.87} C_VEL
LIN {X 0,Y 602.53,Z 123.436,A -85,B 0,C 180,E1 -551.591,E2 -551.591} C_VEL
LIN {X 0,Y 601.476,Z 123.564,A -85,B 0,C 180,E1 -552.147,E2 -552.147} C_VEL
LIN {X 0,Y 601.38,Z 123.572,A -85,B 0,C 180,E1 -552.336,E2 -552.336} C_VEL
LIN {X 0,Y 601.377,Z 123.569,A -85,B 0,C 180,E1 -554.898,E2 -554.898} C_VEL
LIN {X 0,Y 601.376,Z 123.578,A -85,B 0,C 180,E1 -557.688,E2 -557.688} C_VEL
LIN {X 0,Y 601.383,Z 123.578,A -85,B 0,C 180,E1 -559.809,E2 -559.809} C_VEL
LIN {X 0,Y 601.353,Z 123.572,A -85,B 0,C 180,E1 -562.59,E2 -562.59} C_VEL
LIN {X 0,Y 601.378,Z 123.57,A -85,B 0,C 180,E1 -564.879,E2 -564.879} C_VEL
LIN {X 0,Y 601.398,Z 123.573,A -85,B 0,C 180,E1 -567.358,E2 -567.358} C_VEL
LIN {X 0,Y 601.372,Z 123.571,A -85,B 0,C 180,E1 -570.166,E2 -570.166} C_VEL
LIN {X 0,Y 601.387,Z 123.568,A -85,B 0,C 180,E1 -572.709,E2 -572.709} C_VEL
LIN {X 0,Y 601.37,Z 123.576,A -85,B 0,C 180,E1 -575.108,E2 -575.108} C_VEL
LIN {X 0,Y 601.428,Z 123.571,A -85,B 0,C 180,E1 -577.419,E2 -577.419} C_VEL
LIN {X 0,Y 601.373,Z 123.57,A -85,B 0,C 180,E1 -579.997,E2 -579.997} C_VEL
LIN {X 0,Y 601.369,Z 123.572,A -85,B 0,C 180,E1 -582.673,E2 -582.673} C_VEL
LIN {X 0,Y 601.396,Z 123.571,A -85,B 0,C 180,E1 -585.479,E2 -585.479} C_VEL
LIN {X 0,Y 601.401,Z 123.567,A -85,B 0,C 180,E1 -588.408,E2 -588.408} C_VEL
LIN {X 0,Y 601.396,Z 123.575,A -85,B 0,C 180,E1 -590.872,E2 -590.872} C_VEL
LIN {X 0,Y 601.391,Z 123.57,A -85,B 0,C 180,E1 -593.416,E2 -593.416} C_VEL
LIN {X 0,Y 601.392,Z 123.567,A -85,B 0,C 180,E1 -596.069,E2 -596.069} C_VEL
LIN {X 0,Y 601.387,Z 123.574,A -85,B 0,C 180,E1 -599.056,E2 -599.056} C_VEL
LIN {X 0,Y 601.383,Z 123.57,A -85,B 0,C 180,E1 -601.37,E2 -601.37} C_VEL
LIN {X 0,Y 601.367,Z 123.57,A -85,B 0,C 180,E1 -603.634,E2 -603.634} C_VEL
LIN {X 0,Y 601.388,Z 123.568,A -85,B 0,C 180,E1 -605.856,E2 -605.856} C_VEL
LIN {X 0,Y 601.387,Z 123.575,A -85,B 0,C 180,E1 -608.76,E2 -608.76} C_VEL
LIN {X 0,Y 601.354,Z 123.572,A -85,B 0,C 180,E1 -611.606,E2 -611.606} C_VEL
LIN {X 0,Y 601.384,Z 123.578,A -85,B 0,C 180,E1 -614.408,E2 -614.408} C_VEL
LIN {X 0,Y 601.383,Z 123.577,A -85,B 0,C 180,E1 -616.483,E2 -616.483} C_VEL
LIN {X 0,Y 601.349,Z 123.572,A -85,B 0,C 180,E1 -619.222,E2 -619.222} C_VEL
LIN {X 0,Y 601.422,Z 123.568,A -85,B 0,C 180,E1 -621.939,E2 -621.939} C_VEL
LIN {X 0,Y 601.388,Z 123.571,A -85,B 0,C 180,E1 -624.635,E2 -624.635} C_VEL
LIN {X 0,Y 601.388,Z 123.568,A -85,B 0,C 180,E1 -627.321,E2 -627.321} C_VEL
LIN {X 0,Y 601.437,Z 123.572,A -85,B 0,C 180,E1 -630,E2 -630} C_VEL
LIN {X 0,Y 601.39,Z 123.57,A -85,B 0,C 180,E1 -632.679,E2 -632.679} C_VEL
LIN {X 0,Y 601.394,Z 123.716,A -85,B 0,C 180,E1 -633.266,E2 -633.266} C_VEL
LIN {X 0,Y 601.452,Z 139.712,A -85,B 0,C 180,E1 -636.037,E2 -636.037} C_VEL
LIN {X 0,Y 601.382,Z 155.544,A -85,B 0,C 180,E1 -638.738,E2 -638.738} C_VEL
LIN {X 0,Y 601.38,Z 156.418,A -85,B 0,C 180,E1 -638.887,E2 -638.887} C_VEL
LIN {X 0,Y 601.665,Z 167.789,A -85,B 0,C 180,E1 -639.031,E2 -639.031} C_VEL
LIN {X 0,Y 601.565,Z 262.619,A -85,B 0,C 180,E1 -640.178,E2 -640.178} C_VEL
LIN {X 0,Y 601.524,Z 276.01,A -85,B 0,C 180,E1 -640.476,E2 -640.476} C_VEL
LIN {X 0,Y 601.535,Z 288.992,A -85,B 0,C 180,E1 -640.912,E2 -640.912} C_VEL
LIN {X 0,Y 601.523,Z 300.916,A -85,B 0,C 180,E1 -641.456,E2 -641.456} C_VEL
LIN {X 0,Y 601.481,Z 312.505,A -85,B 0,C 180,E1 -642.141,E2 -642.141} C_VEL
LIN {X 0,Y 601.452,Z 322.961,A -85,B 0,C 180,E1 -642.913,E2 -642.913} C_VEL
LIN {X 0,Y 601.401,Z 332.569,A -85,B 0,C 180,E1 -643.792,E2 -643.792} C_VEL
LIN {X 0,Y 601.393,Z 340.858,A -85,B 0,C 180,E1 -644.725,E2 -644.725} C_VEL
LIN {X 0,Y 601.371,Z 348.373,A -85,B 0,C 180,E1 -645.766,E2 -645.766} C_VEL
LIN {X 0,Y 601.359,Z 353.263,A -85,B 0,C 180,E1 -646.603,E2 -646.603} C_VEL
LIN {X 0,Y 601.355,Z 358.376,A -85,B 0,C 180,E1 -647.69,E2 -647.69} C_VEL
LIN {X 0,Y 601.34,Z 362.287,A -85,B 0,C 180,E1 -648.8,E2 -648.8} C_VEL
LIN {X 0,Y 601.316,Z 364.78,A -85,B 0,C 180,E1 -649.812,E2 -649.812} C_VEL
LIN {X 0,Y 601.339,Z 366.268,A -85,B 0,C 180,E1 -650.777,E2 -650.777} C_VEL
LIN {X 0,Y 601.334,Z 366.987,A -85,B 0,C 180,E1 -651.962,E2 -651.962} C_VEL
LIN {X 0,Y 601.316,Z 366.803,A -85,B 0,C 180,E1 -652.687,E2 -652.687} C_VEL
LIN {X 0,Y 601.324,Z 366.15,A -85,B 0,C 180,E1 -653.414,E2 -653.414} C_VEL
LIN {X 0,Y 601.32,Z 364.795,A -85,B 0,C 180,E1 -654.27,E2 -654.27} C_VEL
LIN {X 0,Y 601.336,Z 362.407,A -85,B 0,C 180,E1 -655.251,E2 -655.251} C_VEL
LIN {X 0,Y 601.38,Z 358.526,A -85,B 0,C 180,E1 -656.365,E2 -656.365} C_VEL
LIN {X 0,Y 601.36,Z 352.75,A -85,B 0,C 180,E1 -657.582,E2 -657.582} C_VEL
LIN {X 0,Y 601.37,Z 346.337,A -85,B 0,C 180,E1 -658.63,E2 -658.63} C_VEL
LIN {X 0,Y 601.399,Z 339.07,A -85,B 0,C 180,E1 -659.587,E2 -659.587} C_VEL
LIN {X 0,Y 601.413,Z 329.974,A -85,B 0,C 180,E1 -660.553,E2 -660.553} C_VEL
LIN {X 0,Y 601.455,Z 320.171,A -85,B 0,C 180,E1 -661.4,E2 -661.4} C_VEL
LIN {X 0,Y 601.454,Z 309.933,A -85,B 0,C 180,E1 -662.118,E2 -662.118} C_VEL
LIN {X 0,Y 601.514,Z 298.998,A -85,B 0,C 180,E1 -662.731,E2 -662.731} C_VEL
LIN {X 0,Y 601.554,Z 286.714,A -85,B 0,C 180,E1 -663.265,E2 -663.265} C_VEL
LIN {X 0,Y 601.582,Z 273.631,A -85,B 0,C 180,E1 -663.679,E2 -663.679} C_VEL
LIN {X 0,Y 601.593,Z 261.157,A -85,B 0,C 180,E1 -663.934,E2 -663.934} C_VEL
LIN {X 0,Y 601.534,Z 157.335,A -85,B 0,C 180,E1 -665.188,E2 -665.188} C_VEL
LIN {X 0,Y 601.421,Z 156.378,A -85,B 0,C 180,E1 -665.209,E2 -665.209} C_VEL
LIN {X 0,Y 601.446,Z 140.949,A -85,B 0,C 180,E1 -667.841,E2 -667.841} C_VEL
LIN {X 0,Y 601.506,Z 126.806,A -85,B 0,C 180,E1 -670.282,E2 -670.282} C_VEL
LIN {X 0,Y 601.434,Z 123.565,A -85,B 0,C 180,E1 -670.873,E2 -670.873} C_VEL
LIN {X 0,Y 601.446,Z 123.565,A -85,B 0,C 180,E1 -673.585,E2 -673.585} C_VEL
LIN {X 0,Y 601.446,Z 123.563,A -85,B 0,C 180,E1 -676.426,E2 -676.426} C_VEL
LIN {X 0,Y 601.416,Z 123.569,A -85,B 0,C 180,E1 -679.427,E2 -679.427} C_VEL
LIN {X 0,Y 601.42,Z 123.574,A -85,B 0,C 180,E1 -681.733,E2 -681.733} C_VEL
LIN {X 0,Y 601.382,Z 123.57,A -85,B 0,C 180,E1 -684.246,E2 -684.246} C_VEL
LIN {X 0,Y 601.418,Z 123.564,A -85,B 0,C 180,E1 -686.687,E2 -686.687} C_VEL
LIN {X 0,Y 601.412,Z 123.568,A -85,B 0,C 180,E1 -689.058,E2 -689.058} C_VEL
LIN {X 0,Y 601.432,Z 123.572,A -85,B 0,C 180,E1 -691.374,E2 -691.374} C_VEL
LIN {X 0,Y 601.397,Z 123.572,A -85,B 0,C 180,E1 -693.637,E2 -693.637} C_VEL
LIN {X 0,Y 601.416,Z 123.566,A -85,B 0,C 180,E1 -696.59,E2 -696.59} C_VEL
LIN {X 0,Y 601.421,Z 123.568,A -85,B 0,C 180,E1 -699.479,E2 -699.479} C_VEL
LIN {X 0,Y 601.391,Z 123.568,A -85,B 0,C 180,E1 -702.312,E2 -702.312} C_VEL
LIN {X 0,Y 601.412,Z 123.567,A -85,B 0,C 180,E1 -704.409,E2 -704.409} C_VEL
LIN {X 0,Y 601.407,Z 123.571,A -85,B 0,C 180,E1 -707.172,E2 -707.172} C_VEL
LIN {X 0,Y 601.428,Z 123.563,A -85,B 0,C 180,E1 -709.906,E2 -709.906} C_VEL
LIN {X 0,Y 601.44,Z 123.57,A -85,B 0,C 180,E1 -712.615,E2 -712.615} C_VEL
LIN {X 0,Y 601.395,Z 123.567,A -85,B 0,C 180,E1 -715.308,E2 -715.308} C_VEL
LIN {X 0,Y 601.435,Z 123.564,A -85,B 0,C 180,E1 -717.992,E2 -717.992} C_VEL
LIN {X 0,Y 601.44,Z 123.567,A -85,B 0,C 180,E1 -720.67,E2 -720.67} C_VEL
LIN {X 0,Y 601.373,Z 123.57,A -85,B 0,C 180,E1 -723.35,E2 -723.35} C_VEL
LIN {X 0,Y 601.437,Z 123.568,A -85,B 0,C 180,E1 -726.037,E2 -726.037} C_VEL
LIN {X 0,Y 601.391,Z 123.569,A -85,B 0,C 180,E1 -728.739,E2 -728.739} C_VEL
LIN {X 0,Y 601.388,Z 123.567,A -85,B 0,C 180,E1 -730.992,E2 -730.992} C_VEL
LIN {X 0,Y 601.402,Z 123.569,A -85,B 0,C 180,E1 -733.517,E2 -733.517} C_VEL
LIN {X 0,Y 601.403,Z 123.569,A -85,B 0,C 180,E1 -736.288,E2 -736.288} C_VEL
LIN {X 0,Y 601.403,Z 123.567,A -85,B 0,C 180,E1 -739.1,E2 -739.1} C_VEL
LIN {X 0,Y 601.385,Z 123.574,A -85,B 0,C 180,E1 -741.961,E2 -741.961} C_VEL
LIN {X 0,Y 601.378,Z 123.57,A -85,B 0,C 180,E1 -744.88,E2 -744.88} C_VEL
LIN {X 0,Y 601.397,Z 123.574,A -85,B 0,C 180,E1 -747.359,E2 -747.359} C_VEL
LIN {X 0,Y 601.373,Z 123.57,A -85,B 0,C 180,E1 -750.168,E2 -750.168} C_VEL
LIN {X 0,Y 601.384,Z 123.57,A -85,B 0,C 180,E1 -752.709,E2 -752.709} C_VEL
LIN {X 0,Y 601.363,Z 123.578,A -85,B 0,C 180,E1 -755.107,E2 -755.107} C_VEL
LIN {X 0,Y 601.395,Z 123.573,A -85,B 0,C 180,E1 -757.422,E2 -757.422} C_VEL
LIN {X 0,Y 601.356,Z 123.572,A -85,B 0,C 180,E1 -760,E2 -760} C_VEL
LIN {X 0,Y 601.367,Z 123.576,A -85,B 0,C 180,E1 -762.675,E2 -762.675} C_VEL
LIN {X 0,Y 601.402,Z 123.568,A -85,B 0,C 180,E1 -765.48,E2 -765.48} C_VEL
LIN {X 0,Y 601.405,Z 123.57,A -85,B 0,C 180,E1 -768.409,E2 -768.409} C_VEL
LIN {X 0,Y 601.396,Z 123.575,A -85,B 0,C 180,E1 -770.872,E2 -770.872} C_VEL
LIN {X 0,Y 601.387,Z 123.568,A -85,B 0,C 180,E1 -773.416,E2 -773.416} C_VEL
LIN {X 0,Y 601.413,Z 123.568,A -85,B 0,C 180,E1 -776.068,E2 -776.068} C_VEL
LIN {X 0,Y 601.393,Z 123.569,A -85,B 0,C 180,E1 -779.056,E2 -779.056} C_VEL
LIN {X 0,Y 601.392,Z 123.568,A -85,B 0,C 180,E1 -781.371,E2 -781.371} C_VEL
LIN {X 0,Y 601.41,Z 123.573,A -85,B 0,C 180,E1 -784.134,E2 -784.134} C_VEL
LIN {X 0,Y 601.404,Z 123.57,A -85,B 0,C 180,E1 -787.044,E2 -787.044} C_VEL
LIN {X 0,Y 601.379,Z 123.579,A -85,B 0,C 180,E1 -787.134,E2 -787.134} C_VEL
LIN {X 0,Y 601.667,Z 130.051,A -85,B 0,C 180,E1 -788.051,E2 -788.051} C_VEL
LIN {X 0,Y 601.577,Z 149.468,A -85,B 0,C 180,E1 -790.729,E2 -790.729} C_VEL
LIN {X 0,Y 601.522,Z 169.648,A -85,B 0,C 180,E1 -793.469,E2 -793.469} C_VEL
LIN {X 0,Y 601.475,Z 191.079,A -85,B 0,C 180,E1 -796.338,E2 -796.338} C_VEL
LIN {X 0,Y 601.417,Z 194.613,A -85,B 0,C 180,E1 -796.807,E2 -796.807} C_VEL
LIN {X 0,Y 601.658,Z 198.724,A -85,B 0,C 180,E1 -796.877,E2 -796.877} C_VEL
LIN {X 0,Y 601.614,Z 302.95,A -85,B 0,C 180,E1 -798.14,E2 -798.14} C_VEL
LIN {X 0,Y 601.56,Z 316.22,A -85,B 0,C 180,E1 -798.438,E2 -798.438} C_VEL
LIN {X 0,Y 601.546,Z 327.906,A -85,B 0,C 180,E1 -798.825,E2 -798.825} C_VEL
LIN {X 0,Y 601.522,Z 340.634,A -85,B 0,C 180,E1 -799.396,E2 -799.396} C_VEL
LIN {X 0,Y 601.483,Z 352.2,A -85,B 0,C 180,E1 -800.076,E2 -800.076} C_VEL
LIN {X 0,Y 601.444,Z 362.597,A -85,B 0,C 180,E1 -800.839,E2 -800.839} C_VEL
LIN {X 0,Y 601.429,Z 371.113,A -85,B 0,C 180,E1 -801.601,E2 -801.601} C_VEL
LIN {X 0,Y 601.418,Z 378.961,A -85,B 0,C 180,E1 -802.446,E2 -802.446} C_VEL
LIN {X 0,Y 601.37,Z 386.226,A -85,B 0,C 180,E1 -803.398,E2 -803.398} C_VEL
LIN {X 0,Y 601.372,Z 391.867,A -85,B 0,C 180,E1 -804.299,E2 -804.299} C_VEL
LIN {X 0,Y 601.336,Z 396.95,A -85,B 0,C 180,E1 -805.307,E2 -805.307} C_VEL
LIN {X 0,Y 601.368,Z 400.896,A -85,B 0,C 180,E1 -806.315,E2 -806.315} C_VEL
LIN {X 0,Y 601.325,Z 403.809,A -85,B 0,C 180,E1 -807.321,E2 -807.321} C_VEL
LIN {X 0,Y 601.344,Z 405.202,A -85,B 0,C 180,E1 -807.991,E2 -807.991} C_VEL
LIN {X 0,Y 601.339,Z 406.784,A -85,B 0,C 180,E1 -809.33,E2 -809.33} C_VEL
LIN {X 0,Y 601.335,Z 407,A -85,B 0,C 180,E1 -810,E2 -810} C_VEL
LIN {X 0,Y 601.347,Z 406.184,A -85,B 0,C 180,E1 -811.34,E2 -811.34} C_VEL
LIN {X 0,Y 601.343,Z 405.202,A -85,B 0,C 180,E1 -812.009,E2 -812.009} C_VEL
LIN {X 0,Y 601.325,Z 403.809,A -85,B 0,C 180,E1 -812.68,E2 -812.68} C_VEL
LIN {X 0,Y 601.368,Z 400.896,A -85,B 0,C 180,E1 -813.685,E2 -813.685} C_VEL
LIN {X 0,Y 601.336,Z 396.949,A -85,B 0,C 180,E1 -814.693,E2 -814.693} C_VEL
LIN {X 0,Y 601.373,Z 390.876,A -85,B 0,C 180,E1 -815.869,E2 -815.869} C_VEL
LIN {X 0,Y 601.382,Z 384.234,A -85,B 0,C 180,E1 -816.88,E2 -816.88} C_VEL
LIN {X 0,Y 601.4,Z 375.988,A -85,B 0,C 180,E1 -817.892,E2 -817.892} C_VEL
LIN {X 0,Y 601.436,Z 367.535,A -85,B 0,C 180,E1 -818.738,E2 -818.738} C_VEL
LIN {X 0,Y 601.449,Z 357.09,A -85,B 0,C 180,E1 -819.585,E2 -819.585} C_VEL
LIN {X 0,Y 601.467,Z 346.755,A -85,B 0,C 180,E1 -820.265,E2 -820.265} C_VEL
LIN {X 0,Y 601.538,Z 334.598,A -85,B 0,C 180,E1 -820.896,E2 -820.896} C_VEL
LIN {X 0,Y 601.555,Z 322.212,A -85,B 0,C 180,E1 -821.379,E2 -821.379} C_VEL
LIN {X 0,Y 601.583,Z 309.428,A -85,B 0,C 180,E1 -821.733,E2 -821.733} C_VEL
LIN {X 0,Y 601.62,Z 297.067,A -85,B 0,C 180,E1 -821.946,E2 -821.946} C_VEL
LIN {X 0,Y 601.471,Z 195.123,A -85,B 0,C 180,E1 -823.171,E2 -823.171} C_VEL
LIN {X 0,Y 601.455,Z 194.126,A -85,B 0,C 180,E1 -823.257,E2 -823.257} C_VEL
LIN {X 0,Y 601.519,Z 172.767,A -85,B 0,C 180,E1 -826.111,E2 -826.111} C_VEL
LIN {X 0,Y 601.598,Z 150.761,A -85,B 0,C 180,E1 -829.093,E2 -829.093} C_VEL
LIN {X 0,Y 601.666,Z 130.049,A -85,B 0,C 180,E1 -831.95,E2 -831.95} C_VEL
LIN {X 0,Y 601.379,Z 123.577,A -85,B 0,C 180,E1 -832.866,E2 -832.866} C_VEL
LIN {X 0,Y 601.421,Z 123.572,A -85,B 0,C 180,E1 -835.618,E2 -835.618} C_VEL
LIN {X 0,Y 601.386,Z 123.576,A -85,B 0,C 180,E1 -837.869,E2 -837.869} C_VEL
LIN {X 0,Y 601.403,Z 123.569,A -85,B 0,C 180,E1 -840.166,E2 -840.166} C_VEL
LIN {X 0,Y 601.396,Z 123.567,A -85,B 0,C 180,E1 -842.711,E2 -842.711} C_VEL
LIN {X 0,Y 601.382,Z 123.572,A -85,B 0,C 180,E1 -845.109,E2 -845.109} C_VEL
LIN {X 0,Y 601.435,Z 123.571,A -85,B 0,C 180,E1 -847.419,E2 -847.419} C_VEL
LIN {X 0,Y 601.381,Z 123.57,A -85,B 0,C 180,E1 -849.998,E2 -849.998} C_VEL
LIN {X 0,Y 601.377,Z 123.57,A -85,B 0,C 180,E1 -852.674,E2 -852.674} C_VEL
LIN {X 0,Y 601.404,Z 123.573,A -85,B 0,C 180,E1 -855.479,E2 -855.479} C_VEL
LIN {X 0,Y 601.408,Z 123.565,A -85,B 0,C 180,E1 -858.409,E2 -858.409} C_VEL
LIN {X 0,Y 601.399,Z 123.57,A -85,B 0,C 180,E1 -861.534,E2 -861.534} C_VEL
LIN {X 0,Y 601.39,Z 123.569,A -85,B 0,C 180,E1 -863.742,E2 -863.742} C_VEL
LIN {X 0,Y 601.415,Z 123.569,A -85,B 0,C 180,E1 -866.685,E2 -866.685} C_VEL
LIN {X 0,Y 601.399,Z 123.575,A -85,B 0,C 180,E1 -869.056,E2 -869.056} C_VEL
LIN {X 0,Y 601.4,Z 123.569,A -85,B 0,C 180,E1 -871.371,E2 -871.371} C_VEL
LIN {X 0,Y 601.381,Z 123.569,A -85,B 0,C 180,E1 -873.635,E2 -873.635} C_VEL
LIN {X 0,Y 601.398,Z 123.566,A -85,B 0,C 180,E1 -875.857,E2 -875.857} C_VEL
LIN {X 0,Y 601.397,Z 123.577,A -85,B 0,C 180,E1 -878.76,E2 -878.76} C_VEL
LIN {X 0,Y 601.365,Z 123.57,A -85,B 0,C 180,E1 -881.606,E2 -881.606} C_VEL
LIN {X 0,Y 601.398,Z 123.573,A -85,B 0,C 180,E1 -884.408,E2 -884.408} C_VEL
LIN {X 0,Y 601.365,Z 123.572,A -85,B 0,C 180,E1 -887.17,E2 -887.17} C_VEL
LIN {X 0,Y 601.42,Z 123.566,A -85,B 0,C 180,E1 -889.904,E2 -889.904} C_VEL
LIN {X 0,Y 601.4,Z 123.573,A -85,B 0,C 180,E1 -892.614,E2 -892.614} C_VEL
LIN {X 0,Y 601.379,Z 123.569,A -85,B 0,C 180,E1 -895.307,E2 -895.307} C_VEL
LIN {X 0,Y 601.434,Z 123.567,A -85,B 0,C 180,E1 -897.99,E2 -897.99} C_VEL
LIN {X 0,Y 601.4,Z 123.569,A -85,B 0,C 180,E1 -900.669,E2 -900.669} C_VEL
LIN {X 0,Y 601.408,Z 123.568,A -85,B 0,C 180,E1 -902.679,E2 -902.679} C_VEL
LIN {X 0,Y 601.392,Z 123.568,A -85,B 0,C 180,E1 -905.364,E2 -905.364} C_VEL
LIN {X 0,Y 601.434,Z 123.572,A -85,B 0,C 180,E1 -908.06,E2 -908.06} C_VEL
LIN {X 0,Y 601.381,Z 123.568,A -85,B 0,C 180,E1 -910.988,E2 -910.988} C_VEL
LIN {X 0,Y 601.38,Z 123.572,A -85,B 0,C 180,E1 -912.336,E2 -912.336} C_VEL
LIN {X 0,Y 600.689,Z 123.657,A -85,B 0,C 180,E1 -912.895,E2 -912.895} C_VEL
LIN {X 0,Y 597.833,Z 124.019,A -85,B 0,C 180,E1 -913.803,E2 -913.803} C_VEL
LIN {X 0,Y 595.437,Z 124.313,A -85,B 0,C 180,E1 -914.533,E2 -914.533} C_VEL
LIN {X 0,Y 594.41,Z 124.438,A -85,B 0,C 180,E1 -915.097,E2 -915.097} C_VEL
LIN {X 0,Y 594.326,Z 124.449,A -85,B 0,C 180,E1 -915.288,E2 -915.288} C_VEL
LIN {X 0,Y 594.326,Z 124.456,A -85,B 0,C 180,E1 -917.905,E2 -917.905} C_VEL
LIN {X 0,Y 594.372,Z 124.442,A -85,B 0,C 180,E1 -920.776,E2 -920.776} C_VEL
LIN {X 0,Y 594.346,Z 124.455,A -85,B 0,C 180,E1 -923.705,E2 -923.705} C_VEL
LIN {X 0,Y 594.352,Z 124.448,A -85,B 0,C 180,E1 -926.015,E2 -926.015} C_VEL
LIN {X 0,Y 594.338,Z 124.448,A -85,B 0,C 180,E1 -929,E2 -929} C_VEL
LIN {X 0,Y 594.365,Z 124.45,A -85,B 0,C 180,E1 -931.64,E2 -931.64} C_VEL
LIN {X 0,Y 594.355,Z 124.444,A -85,B 0,C 180,E1 -934.134,E2 -934.134} C_VEL
LIN {X 0,Y 594.374,Z 124.447,A -85,B 0,C 180,E1 -937.087,E2 -937.087} C_VEL
LIN {X 0,Y 594.334,Z 124.449,A -85,B 0,C 180,E1 -939.769,E2 -939.769} C_VEL
LIN {X 0,Y 594.329,Z 124.447,A -85,B 0,C 180,E1 -942.378,E2 -942.378} C_VEL
LIN {X 0,Y 594.334,Z 124.456,A -85,B 0,C 180,E1 -945.193,E2 -945.193} C_VEL
LIN {X 0,Y 594.353,Z 124.444,A -85,B 0,C 180,E1 -948.154,E2 -948.154} C_VEL
LIN {X 0,Y 594.358,Z 124.448,A -85,B 0,C 180,E1 -951.298,E2 -951.298} C_VEL
LIN {X 0,Y 594.333,Z 124.447,A -85,B 0,C 180,E1 -953.754,E2 -953.754} C_VEL
LIN {X 0,Y 594.344,Z 124.447,A -85,B 0,C 180,E1 -956.236,E2 -956.236} C_VEL
LIN {X 0,Y 594.339,Z 124.453,A -85,B 0,C 180,E1 -958.648,E2 -958.648} C_VEL
LIN {X 0,Y 594.363,Z 124.448,A -85,B 0,C 180,E1 -961.044,E2 -961.044} C_VEL
LIN {X 0,Y 594.342,Z 124.446,A -85,B 0,C 180,E1 -963.984,E2 -963.984} C_VEL
LIN {X 0,Y 594.336,Z 124.451,A -85,B 0,C 180,E1 -966.293,E2 -966.293} C_VEL
LIN {X 0,Y 594.364,Z 124.444,A -85,B 0,C 180,E1 -969.223,E2 -969.223} C_VEL
LIN {X 0,Y 594.315,Z 124.453,A -85,B 0,C 180,E1 -972.094,E2 -972.094} C_VEL
LIN {X 0,Y 594.326,Z 124.45,A -85,B 0,C 180,E1 -974.921,E2 -974.921} C_VEL
LIN {X 0,Y 594.355,Z 124.445,A -85,B 0,C 180,E1 -977.711,E2 -977.711} C_VEL
LIN {X 0,Y 594.338,Z 124.453,A -85,B 0,C 180,E1 -980.471,E2 -980.471} C_VEL
LIN {X 0,Y 594.331,Z 124.447,A -85,B 0,C 180,E1 -983.209,E2 -983.209} C_VEL
LIN {X 0,Y 594.342,Z 124.452,A -85,B 0,C 180,E1 -985.931,E2 -985.931} C_VEL
LIN {X 0,Y 594.333,Z 124.449,A -85,B 0,C 180,E1 -988.645,E2 -988.645} C_VEL
LIN {X 0,Y 594.315,Z 124.451,A -85,B 0,C 180,E1 -990.677,E2 -990.677} C_VEL
LIN {X 0,Y 594.358,Z 124.446,A -85,B 0,C 180,E1 -992.711,E2 -992.711} C_VEL
LIN {X 0,Y 594.329,Z 124.527,A -85,B 0,C 180,E1 -993.177,E2 -993.177} C_VEL
LIN {X 0,Y 594.437,Z 137.328,A -85,B 0,C 180,E1 -995.427,E2 -995.427} C_VEL
LIN {X 0,Y 594.36,Z 153.098,A -85,B 0,C 180,E1 -998.157,E2 -998.157} C_VEL
LIN {X 0,Y 594.338,Z 156.339,A -85,B 0,C 180,E1 -998.714,E2 -998.714} C_VEL
LIN {X 0,Y 594.759,Z 160.946,A -85,B 0,C 180,E1 -998.794,E2 -998.794} C_VEL
LIN {X 0,Y 594.629,Z 262.759,A -85,B 0,C 180,E1 -1000.04,E2 -1000.04} C_VEL
LIN {X 0,Y 594.563,Z 276.12,A -85,B 0,C 180,E1 -1000.342,E2 -1000.342} C_VEL
LIN {X 0,Y 594.561,Z 288.819,A -85,B 0,C 180,E1 -1000.773,E2 -1000.773} C_VEL
LIN {X 0,Y 594.535,Z 300.087,A -85,B 0,C 180,E1 -1001.286,E2 -1001.286} C_VEL
LIN {X 0,Y 594.449,Z 311.281,A -85,B 0,C 180,E1 -1001.941,E2 -1001.941} C_VEL
LIN {X 0,Y 594.418,Z 321.938,A -85,B 0,C 180,E1 -1002.721,E2 -1002.721} C_VEL
LIN {X 0,Y 594.393,Z 330.684,A -85,B 0,C 180,E1 -1003.504,E2 -1003.504} C_VEL
LIN {X 0,Y 594.346,Z 338.77,A -85,B 0,C 180,E1 -1004.378,E2 -1004.378} C_VEL
LIN {X 0,Y 594.302,Z 346.664,A -85,B 0,C 180,E1 -1005.431,E2 -1005.431} C_VEL
LIN {X 0,Y 594.27,Z 353.003,A -85,B 0,C 180,E1 -1006.489,E2 -1006.489} C_VEL
LIN {X 0,Y 594.278,Z 358.017,A -85,B 0,C 180,E1 -1007.552,E2 -1007.552} C_VEL
LIN {X 0,Y 594.251,Z 361.854,A -85,B 0,C 180,E1 -1008.622,E2 -1008.622} C_VEL
LIN {X 0,Y 594.214,Z 363.825,A -85,B 0,C 180,E1 -1009.34,E2 -1009.34} C_VEL
LIN {X 0,Y 594.219,Z 365.28,A -85,B 0,C 180,E1 -1010.059,E2 -1010.059} C_VEL
LIN {X 0,Y 594.247,Z 366.41,A -85,B 0,C 180,E1 -1010.885,E2 -1010.885} C_VEL
LIN {X 0,Y 594.224,Z 366.876,A -85,B 0,C 180,E1 -1011.509,E2 -1011.509} C_VEL
LIN {X 0,Y 594.237,Z 366.794,A -85,B 0,C 180,E1 -1012.708,E2 -1012.708} C_VEL
LIN {X 0,Y 594.224,Z 365.798,A -85,B 0,C 180,E1 -1013.711,E2 -1013.711} C_VEL
LIN {X 0,Y 594.235,Z 364.465,A -85,B 0,C 180,E1 -1014.453,E2 -1014.453} C_VEL
LIN {X 0,Y 594.241,Z 361.523,A -85,B 0,C 180,E1 -1015.574,E2 -1015.574} C_VEL
LIN {X 0,Y 594.28,Z 357.322,A -85,B 0,C 180,E1 -1016.705,E2 -1016.705} C_VEL
LIN {X 0,Y 594.286,Z 351.682,A -85,B 0,C 180,E1 -1017.847,E2 -1017.847} C_VEL
LIN {X 0,Y 594.307,Z 344.27,A -85,B 0,C 180,E1 -1019.002,E2 -1019.002} C_VEL
LIN {X 0,Y 594.33,Z 336.664,A -85,B 0,C 180,E1 -1019.954,E2 -1019.954} C_VEL
LIN {X 0,Y 594.379,Z 327.885,A -85,B 0,C 180,E1 -1020.855,E2 -1020.855} C_VEL
LIN {X 0,Y 594.448,Z 317.556,A -85,B 0,C 180,E1 -1021.71,E2 -1021.71} C_VEL
LIN {X 0,Y 594.468,Z 306.594,A -85,B 0,C 180,E1 -1022.442,E2 -1022.442} C_VEL
LIN {X 0,Y 594.539,Z 295.254,A -85,B 0,C 180,E1 -1023.041,E2 -1023.041} C_VEL
LIN {X 0,Y 594.594,Z 282.663,A -85,B 0,C 180,E1 -1023.544,E2 -1023.544} C_VEL
LIN {X 0,Y 594.642,Z 269.814,A -85,B 0,C 180,E1 -1023.908,E2 -1023.908} C_VEL
LIN {X 0,Y 594.659,Z 256.701,A -85,B 0,C 180,E1 -1024.138,E2 -1024.138} C_VEL
LIN {X 0,Y 594.667,Z 158.262,A -85,B 0,C 180,E1 -1025.331,E2 -1025.331} C_VEL
LIN {X 0,Y 594.401,Z 156.37,A -85,B 0,C 180,E1 -1025.369,E2 -1025.369} C_VEL
LIN {X 0,Y 594.438,Z 140.384,A -85,B 0,C 180,E1 -1028.13,E2 -1028.13} C_VEL
LIN {X 0,Y 594.464,Z 124.953,A -85,B 0,C 180,E1 -1030.833,E2 -1030.833} C_VEL
LIN {X 0,Y 594.381,Z 124.444,A -85,B 0,C 180,E1 -1030.988,E2 -1030.988} C_VEL
LIN {X 0,Y 594.379,Z 124.449,A -85,B 0,C 180,E1 -1033.842,E2 -1033.842} C_VEL
LIN {X 0,Y 594.377,Z 124.442,A -85,B 0,C 180,E1 -1036.702,E2 -1036.702} C_VEL
LIN {X 0,Y 594.371,Z 124.446,A -85,B 0,C 180,E1 -1039.434,E2 -1039.434} C_VEL
LIN {X 0,Y 594.389,Z 124.441,A -85,B 0,C 180,E1 -1042.392,E2 -1042.392} C_VEL
LIN {X 0,Y 594.379,Z 124.448,A -85,B 0,C 180,E1 -1045.421,E2 -1045.421} C_VEL
LIN {X 0,Y 594.376,Z 124.442,A -85,B 0,C 180,E1 -1048.358,E2 -1048.358} C_VEL
LIN {X 0,Y 594.383,Z 124.444,A -85,B 0,C 180,E1 -1051.043,E2 -1051.043} C_VEL
LIN {X 0,Y 594.38,Z 124.442,A -85,B 0,C 180,E1 -1053.979,E2 -1053.979} C_VEL
LIN {X 0,Y 594.382,Z 124.441,A -85,B 0,C 180,E1 -1056.296,E2 -1056.296} C_VEL
LIN {X 0,Y 594.4,Z 124.447,A -85,B 0,C 180,E1 -1059.225,E2 -1059.225} C_VEL
LIN {X 0,Y 594.342,Z 124.446,A -85,B 0,C 180,E1 -1062.095,E2 -1062.095} C_VEL
LIN {X 0,Y 594.362,Z 124.444,A -85,B 0,C 180,E1 -1064.22,E2 -1064.22} C_VEL
LIN {X 0,Y 594.357,Z 124.451,A -85,B 0,C 180,E1 -1067.017,E2 -1067.017} C_VEL
LIN {X 0,Y 594.386,Z 124.44,A -85,B 0,C 180,E1 -1069.785,E2 -1069.785} C_VEL
LIN {X 0,Y 594.393,Z 124.446,A -85,B 0,C 180,E1 -1072.527,E2 -1072.527} C_VEL
LIN {X 0,Y 594.369,Z 124.443,A -85,B 0,C 180,E1 -1075.253,E2 -1075.253} C_VEL
LIN {X 0,Y 594.403,Z 124.44,A -85,B 0,C 180,E1 -1077.968,E2 -1077.968} C_VEL
LIN {X 0,Y 594.412,Z 124.442,A -85,B 0,C 180,E1 -1080.678,E2 -1080.678} C_VEL
LIN {X 0,Y 594.391,Z 124.444,A -85,B 0,C 180,E1 -1082.711,E2 -1082.711} C_VEL
LIN {X 0,Y 594.372,Z 124.441,A -85,B 0,C 180,E1 -1085.428,E2 -1085.428} C_VEL
LIN {X 0,Y 594.38,Z 124.451,A -85,B 0,C 180,E1 -1088.158,E2 -1088.158} C_VEL
LIN {X 0,Y 594.367,Z 124.441,A -85,B 0,C 180,E1 -1091.061,E2 -1091.061} C_VEL
LIN {X 0,Y 594.372,Z 124.447,A -85,B 0,C 180,E1 -1093.68,E2 -1093.68} C_VEL
LIN {X 0,Y 594.329,Z 124.447,A -85,B 0,C 180,E1 -1096.697,E2 -1096.697} C_VEL
LIN {X 0,Y 594.355,Z 124.447,A -85,B 0,C 180,E1 -1099.335,E2 -1099.335} C_VEL
LIN {X 0,Y 594.349,Z 124.451,A -85,B 0,C 180,E1 -1101.504,E2 -1101.504} C_VEL
LIN {X 0,Y 594.344,Z 124.446,A -85,B 0,C 180,E1 -1104.449,E2 -1104.449} C_VEL
LIN {X 0,Y 594.351,Z 124.444,A -85,B 0,C 180,E1 -1106.702,E2 -1106.702} C_VEL
LIN {X 0,Y 594.336,Z 124.45,A -85,B 0,C 180,E1 -1109.779,E2 -1109.779} C_VEL
LIN {X 0,Y 594.333,Z 124.447,A -85,B 0,C 180,E1 -1112.15,E2 -1112.15} C_VEL
LIN {X 0,Y 594.329,Z 124.448,A -85,B 0,C 180,E1 -1114.584,E2 -1114.584} C_VEL
LIN {X 0,Y 594.351,Z 124.448,A -85,B 0,C 180,E1 -1117.603,E2 -1117.603} C_VEL
LIN {X 0,Y 594.339,Z 124.449,A -85,B 0,C 180,E1 -1120.57,E2 -1120.57} C_VEL
LIN {X 0,Y 594.34,Z 124.451,A -85,B 0,C 180,E1 -1123.302,E2 -1123.302} C_VEL
LIN {X 0,Y 594.344,Z 124.447,A -85,B 0,C 180,E1 -1126.163,E2 -1126.163} C_VEL
LIN {X 0,Y 594.359,Z 124.447,A -85,B 0,C 180,E1 -1129.181,E2 -1129.181} C_VEL
LIN {X 0,Y 594.348,Z 124.446,A -85,B 0,C 180,E1 -1132.056,E2 -1132.056} C_VEL
LIN {X 0,Y 594.32,Z 124.457,A -85,B 0,C 180,E1 -1134.681,E2 -1134.681} C_VEL
LIN {X 0,Y 594.371,Z 124.444,A -85,B 0,C 180,E1 -1137.09,E2 -1137.09} C_VEL
LIN {X 0,Y 594.366,Z 124.444,A -85,B 0,C 180,E1 -1139.676,E2 -1139.676} C_VEL
LIN {X 0,Y 594.361,Z 124.45,A -85,B 0,C 180,E1 -1142.538,E2 -1142.538} C_VEL
LIN {X 0,Y 594.369,Z 124.446,A -85,B 0,C 180,E1 -1144.807,E2 -1144.807} C_VEL
LIN {X 0,Y 594.389,Z 124.55,A -85,B 0,C 180,E1 -1146.988,E2 -1146.988} C_VEL
LIN {X 0,Y 594.758,Z 129.044,A -85,B 0,C 180,E1 -1147.64,E2 -1147.64} C_VEL
LIN {X 0,Y 594.662,Z 149.468,A -85,B 0,C 180,E1 -1150.496,E2 -1150.496} C_VEL
LIN {X 0,Y 594.548,Z 171.474,A -85,B 0,C 180,E1 -1153.519,E2 -1153.519} C_VEL
LIN {X 0,Y 594.425,Z 193.481,A -85,B 0,C 180,E1 -1156.496,E2 -1156.496} C_VEL
LIN {X 0,Y 594.436,Z 194.613,A -85,B 0,C 180,E1 -1156.649,E2 -1156.649} C_VEL
LIN {X 0,Y 594.74,Z 198.724,A -85,B 0,C 180,E1 -1156.721,E2 -1156.721} C_VEL
LIN {X 0,Y 594.666,Z 302.95,A -85,B 0,C 180,E1 -1157.999,E2 -1157.999} C_VEL
LIN {X 0,Y 594.601,Z 316.221,A -85,B 0,C 180,E1 -1158.3,E2 -1158.3} C_VEL
LIN {X 0,Y 594.577,Z 328.49,A -85,B 0,C 180,E1 -1158.715,E2 -1158.715} C_VEL
LIN {X 0,Y 594.536,Z 340.633,A -85,B 0,C 180,E1 -1159.27,E2 -1159.27} C_VEL
LIN {X 0,Y 594.477,Z 352.202,A -85,B 0,C 180,E1 -1159.958,E2 -1159.958} C_VEL
LIN {X 0,Y 594.414,Z 362.598,A -85,B 0,C 180,E1 -1160.73,E2 -1160.73} C_VEL
LIN {X 0,Y 594.383,Z 371.113,A -85,B 0,C 180,E1 -1161.501,E2 -1161.501} C_VEL
LIN {X 0,Y 594.347,Z 378.961,A -85,B 0,C 180,E1 -1162.355,E2 -1162.355} C_VEL
LIN {X 0,Y 594.283,Z 386.815,A -85,B 0,C 180,E1 -1163.409,E2 -1163.409} C_VEL
LIN {X 0,Y 594.289,Z 393.681,A -85,B 0,C 180,E1 -1164.571,E2 -1164.571} C_VEL
LIN {X 0,Y 594.27,Z 398.372,A -85,B 0,C 180,E1 -1165.591,E2 -1165.591} C_VEL
LIN {X 0,Y 594.267,Z 401.957,A -85,B 0,C 180,E1 -1166.61,E2 -1166.61} C_VEL
LIN {X 0,Y 594.226,Z 403.809,A -85,B 0,C 180,E1 -1167.289,E2 -1167.289} C_VEL
LIN {X 0,Y 594.242,Z 405.201,A -85,B 0,C 180,E1 -1167.967,E2 -1167.967} C_VEL
LIN {X 0,Y 594.239,Z 406.784,A -85,B 0,C 180,E1 -1169.322,E2 -1169.322} C_VEL
LIN {X 0,Y 594.236,Z 407,A -85,B 0,C 180,E1 -1170,E2 -1170} C_VEL
LIN {X 0,Y 594.247,Z 406.185,A -85,B 0,C 180,E1 -1171.356,E2 -1171.356} C_VEL
LIN {X 0,Y 594.242,Z 405.201,A -85,B 0,C 180,E1 -1172.033,E2 -1172.033} C_VEL
LIN {X 0,Y 594.226,Z 403.809,A -85,B 0,C 180,E1 -1172.712,E2 -1172.712} C_VEL
LIN {X 0,Y 594.289,Z 400.895,A -85,B 0,C 180,E1 -1173.729,E2 -1173.729} C_VEL
LIN {X 0,Y 594.241,Z 396.949,A -85,B 0,C 180,E1 -1174.749,E2 -1174.749} C_VEL
LIN {X 0,Y 594.305,Z 390.876,A -85,B 0,C 180,E1 -1175.939,E2 -1175.939} C_VEL
LIN {X 0,Y 594.308,Z 384.235,A -85,B 0,C 180,E1 -1176.962,E2 -1176.962} C_VEL
LIN {X 0,Y 594.359,Z 375.988,A -85,B 0,C 180,E1 -1177.987,E2 -1177.987} C_VEL
LIN {X 0,Y 594.382,Z 367.535,A -85,B 0,C 180,E1 -1178.842,E2 -1178.842} C_VEL
LIN {X 0,Y 594.432,Z 357.092,A -85,B 0,C 180,E1 -1179.7,E2 -1179.7} C_VEL
LIN {X 0,Y 594.482,Z 346.755,A -85,B 0,C 180,E1 -1180.387,E2 -1180.387} C_VEL
LIN {X 0,Y 594.558,Z 335.728,A -85,B 0,C 180,E1 -1180.973,E2 -1180.973} C_VEL
LIN {X 0,Y 594.579,Z 323.707,A -85,B 0,C 180,E1 -1181.464,E2 -1181.464} C_VEL
LIN {X 0,Y 594.625,Z 310.341,A -85,B 0,C 180,E1 -1181.851,E2 -1181.851} C_VEL
LIN {X 0,Y 594.7,Z 297.067,A -85,B 0,C 180,E1 -1182.087,E2 -1182.087} C_VEL
LIN {X 0,Y 594.618,Z 196.242,A -85,B 0,C 180,E1 -1183.312,E2 -1183.312} C_VEL
LIN {X 0,Y 594.436,Z 194.611,A -85,B 0,C 180,E1 -1183.351,E2 -1183.351} C_VEL
LIN {X 0,Y 594.518,Z 172.767,A -85,B 0,C 180,E1 -1186.306,E2 -1186.306} C_VEL
LIN {X 0,Y 594.63,Z 152.407,A -85,B 0,C 180,E1 -1189.098,E2 -1189.098} C_VEL
LIN {X 0,Y 594.752,Z 131.344,A -85,B 0,C 180,E1 -1192.036,E2 -1192.036} C_VEL
LIN {X 0,Y 594.624,Z 126.02,A -85,B 0,C 180,E1 -1192.794,E2 -1192.794} C_VEL
LIN {X 0,Y 594.377,Z 124.446,A -85,B 0,C 180,E1 -1193.059,E2 -1193.059} C_VEL
LIN {X 0,Y 594.361,Z 124.45,A -85,B 0,C 180,E1 -1196.017,E2 -1196.017} C_VEL
LIN {X 0,Y 594.332,Z 124.449,A -85,B 0,C 180,E1 -1198.23,E2 -1198.23} C_VEL
LIN {X 0,Y 594.365,Z 124.443,A -85,B 0,C 180,E1 -1200.561,E2 -1200.561} C_VEL
LIN {X 0,Y 594.374,Z 124.443,A -85,B 0,C 180,E1 -1202.951,E2 -1202.951} C_VEL
LIN {X 0,Y 594.327,Z 124.455,A -85,B 0,C 180,E1 -1205.411,E2 -1205.411} C_VEL
LIN {X 0,Y 594.369,Z 124.445,A -85,B 0,C 180,E1 -1207.942,E2 -1207.942} C_VEL
LIN {X 0,Y 594.366,Z 124.444,A -85,B 0,C 180,E1 -1210.82,E2 -1210.82} C_VEL
LIN {X 0,Y 594.348,Z 124.447,A -85,B 0,C 180,E1 -1213.837,E2 -1213.837} C_VEL
LIN {X 0,Y 594.348,Z 124.447,A -85,B 0,C 180,E1 -1216.698,E2 -1216.698} C_VEL
LIN {X 0,Y 594.362,Z 124.449,A -85,B 0,C 180,E1 -1219.432,E2 -1219.432} C_VEL
LIN {X 0,Y 594.385,Z 124.441,A -85,B 0,C 180,E1 -1222.393,E2 -1222.393} C_VEL
LIN {X 0,Y 594.37,Z 124.446,A -85,B 0,C 180,E1 -1225.419,E2 -1225.419} C_VEL
LIN {X 0,Y 594.345,Z 124.445,A -85,B 0,C 180,E1 -1227.851,E2 -1227.851} C_VEL
LIN {X 0,Y 594.34,Z 124.446,A -85,B 0,C 180,E1 -1230.221,E2 -1230.221} C_VEL
LIN {X 0,Y 594.376,Z 124.445,A -85,B 0,C 180,E1 -1233.3,E2 -1233.3} C_VEL
LIN {X 0,Y 594.346,Z 124.447,A -85,B 0,C 180,E1 -1236.294,E2 -1236.294} C_VEL
LIN {X 0,Y 594.379,Z 124.443,A -85,B 0,C 180,E1 -1239.223,E2 -1239.223} C_VEL
LIN {X 0,Y 594.329,Z 124.449,A -85,B 0,C 180,E1 -1242.094,E2 -1242.094} C_VEL
LIN {X 0,Y 594.341,Z 124.45,A -85,B 0,C 180,E1 -1244.921,E2 -1244.921} C_VEL
LIN {X 0,Y 594.347,Z 124.445,A -85,B 0,C 180,E1 -1247.71,E2 -1247.71} C_VEL
LIN {X 0,Y 594.352,Z 124.455,A -85,B 0,C 180,E1 -1250.471,E2 -1250.471} C_VEL
LIN {X 0,Y 594.346,Z 124.445,A -85,B 0,C 180,E1 -1253.208,E2 -1253.208} C_VEL
LIN {X 0,Y 594.35,Z 124.448,A -85,B 0,C 180,E1 -1255.931,E2 -1255.931} C_VEL
LIN {X 0,Y 594.351,Z 124.448,A -85,B 0,C 180,E1 -1258.644,E2 -1258.644} C_VEL
LIN {X 0,Y 594.354,Z 124.447,A -85,B 0,C 180,E1 -1260.677,E2 -1260.677} C_VEL
LIN {X 0,Y 594.375,Z 124.443,A -85,B 0,C 180,E1 -1262.71,E2 -1262.71} C_VEL
LIN {X 0,Y 594.362,Z 124.444,A -85,B 0,C 180,E1 -1265.427,E2 -1265.427} C_VEL
LIN {X 0,Y 594.376,Z 124.449,A -85,B 0,C 180,E1 -1268.157,E2 -1268.157} C_VEL
LIN {X 0,Y 594.349,Z 124.444,A -85,B 0,C 180,E1 -1271.051,E2 -1271.051} C_VEL
LIN {X 0,Y 594.367,Z 124.449,A -85,B 0,C 180,E1 -1273.679,E2 -1273.679} C_VEL
LIN {X 0,Y 594.326,Z 124.449,A -85,B 0,C 180,E1 -1275.288,E2 -1275.288} C_VEL
LIN {X 0,Y 593.656,Z 124.541,A -85,B 0,C 180,E1 -1275.853,E2 -1275.853} C_VEL
LIN {X 0,Y 590.792,Z 124.898,A -85,B 0,C 180,E1 -1276.771,E2 -1276.771} C_VEL
LIN {X 0,Y 588.381,Z 125.197,A -85,B 0,C 180,E1 -1277.509,E2 -1277.509} C_VEL
LIN {X 0,Y 587.356,Z 125.321,A -85,B 0,C 180,E1 -1278.079,E2 -1278.079} C_VEL
LIN {X 0,Y 587.278,Z 125.328,A -85,B 0,C 180,E1 -1278.272,E2 -1278.272} C_VEL
LIN {X 0,Y 587.299,Z 125.324,A -85,B 0,C 180,E1 -1281.038,E2 -1281.038} C_VEL
LIN {X 0,Y 587.286,Z 125.329,A -85,B 0,C 180,E1 -1284.008,E2 -1284.008} C_VEL
LIN {X 0,Y 587.298,Z 125.324,A -85,B 0,C 180,E1 -1286.28,E2 -1286.28} C_VEL
LIN {X 0,Y 587.299,Z 125.326,A -85,B 0,C 180,E1 -1289.124,E2 -1289.124} C_VEL
LIN {X 0,Y 587.313,Z 125.325,A -85,B 0,C 180,E1 -1291.83,E2 -1291.83} C_VEL
LIN {X 0,Y 587.325,Z 125.32,A -85,B 0,C 180,E1 -1294.344,E2 -1294.344} C_VEL
LIN {X 0,Y 587.329,Z 125.324,A -85,B 0,C 180,E1 -1297.608,E2 -1297.608} C_VEL
LIN {X 0,Y 587.289,Z 125.324,A -85,B 0,C 180,E1 -1300.255,E2 -1300.255} C_VEL
LIN {X 0,Y 587.285,Z 125.334,A -85,B 0,C 180,E1 -1303.115,E2 -1303.115} C_VEL
LIN {X 0,Y 587.293,Z 125.323,A -85,B 0,C 180,E1 -1306.046,E2 -1306.046} C_VEL
LIN {X 0,Y 587.305,Z 125.33,A -85,B 0,C 180,E1 -1308.927,E2 -1308.927} C_VEL
LIN {X 0,Y 587.306,Z 125.324,A -85,B 0,C 180,E1 -1311.518,E2 -1311.518} C_VEL
LIN {X 0,Y 587.268,Z 125.327,A -85,B 0,C 180,E1 -1314.098,E2 -1314.098} C_VEL
LIN {X 0,Y 587.325,Z 125.329,A -85,B 0,C 180,E1 -1316.889,E2 -1316.889} C_VEL
LIN {X 0,Y 587.287,Z 125.324,A -85,B 0,C 180,E1 -1319.827,E2 -1319.827} C_VEL
LIN {X 0,Y 587.289,Z 125.328,A -85,B 0,C 180,E1 -1322.317,E2 -1322.317} C_VEL
LIN {X 0,Y 587.29,Z 125.326,A -85,B 0,C 180,E1 -1325.238,E2 -1325.238} C_VEL
LIN {X 0,Y 587.289,Z 125.328,A -85,B 0,C 180,E1 -1328.224,E2 -1328.224} C_VEL
LIN {X 0,Y 587.313,Z 125.322,A -85,B 0,C 180,E1 -1331.15,E2 -1331.15} C_VEL
LIN {X 0,Y 587.279,Z 125.329,A -85,B 0,C 180,E1 -1334.023,E2 -1334.023} C_VEL
LIN {X 0,Y 587.325,Z 125.326,A -85,B 0,C 180,E1 -1336.153,E2 -1336.153} C_VEL
LIN {X 0,Y 587.29,Z 125.325,A -85,B 0,C 180,E1 -1338.961,E2 -1338.961} C_VEL
LIN {X 0,Y 587.319,Z 125.323,A -85,B 0,C 180,E1 -1341.744,E2 -1341.744} C_VEL
LIN {X 0,Y 587.326,Z 125.324,A -85,B 0,C 180,E1 -1344.507,E2 -1344.507} C_VEL
LIN {X 0,Y 587.325,Z 125.32,A -85,B 0,C 180,E1 -1347.256,E2 -1347.256} C_VEL
LIN {X 0,Y 587.373,Z 125.324,A -85,B 0,C 180,E1 -1350,E2 -1350} C_VEL
LIN {X 0,Y 587.326,Z 125.323,A -85,B 0,C 180,E1 -1352.743,E2 -1352.743} C_VEL
LIN {X 0,Y 587.289,Z 125.333,A -85,B 0,C 180,E1 -1353.087,E2 -1353.087} C_VEL
LIN {X 0,Y 587.384,Z 136.912,A -85,B 0,C 180,E1 -1355.148,E2 -1355.148} C_VEL
LIN {X 0,Y 587.32,Z 152.651,A -85,B 0,C 180,E1 -1357.91,E2 -1357.91} C_VEL
LIN {X 0,Y 587.288,Z 156.387,A -85,B 0,C 180,E1 -1358.559,E2 -1358.559} C_VEL
LIN {X 0,Y 587.867,Z 161.13,A -85,B 0,C 180,E1 -1358.638,E2 -1358.638} C_VEL
LIN {X 0,Y 587.703,Z 262.88,A -85,B 0,C 180,E1 -1359.898,E2 -1359.898} C_VEL
LIN {X 0,Y 587.617,Z 276.213,A -85,B 0,C 180,E1 -1360.204,E2 -1360.204} C_VEL
LIN {X 0,Y 587.609,Z 288.885,A -85,B 0,C 180,E1 -1360.64,E2 -1360.64} C_VEL
LIN {X 0,Y 587.543,Z 300.387,A -85,B 0,C 180,E1 -1361.173,E2 -1361.173} C_VEL
LIN {X 0,Y 587.431,Z 311.338,A -85,B 0,C 180,E1 -1361.823,E2 -1361.823} C_VEL
LIN {X 0,Y 587.407,Z 321.978,A -85,B 0,C 180,E1 -1362.612,E2 -1362.612} C_VEL
LIN {X 0,Y 587.339,Z 331.624,A -85,B 0,C 180,E1 -1363.493,E2 -1363.493} C_VEL
LIN {X 0,Y 587.29,Z 340.913,A -85,B 0,C 180,E1 -1364.555,E2 -1364.555} C_VEL
LIN {X 0,Y 587.199,Z 348.426,A -85,B 0,C 180,E1 -1365.622,E2 -1365.622} C_VEL
LIN {X 0,Y 587.192,Z 354.761,A -85,B 0,C 180,E1 -1366.766,E2 -1366.766} C_VEL
LIN {X 0,Y 587.179,Z 359.115,A -85,B 0,C 180,E1 -1367.771,E2 -1367.771} C_VEL
LIN {X 0,Y 587.147,Z 363.003,A -85,B 0,C 180,E1 -1368.987,E2 -1368.987} C_VEL
LIN {X 0,Y 587.149,Z 365.723,A -85,B 0,C 180,E1 -1370.311,E2 -1370.311} C_VEL
LIN {X 0,Y 587.163,Z 366.568,A -85,B 0,C 180,E1 -1371.044,E2 -1371.044} C_VEL
LIN {X 0,Y 587.139,Z 366.946,A -85,B 0,C 180,E1 -1371.781,E2 -1371.781} C_VEL
LIN {X 0,Y 587.124,Z 366.721,A -85,B 0,C 180,E1 -1372.825,E2 -1372.825} C_VEL
LIN {X 0,Y 587.124,Z 365.342,A -85,B 0,C 180,E1 -1374.016,E2 -1374.016} C_VEL
LIN {X 0,Y 587.143,Z 362.891,A -85,B 0,C 180,E1 -1375.146,E2 -1375.146} C_VEL
LIN {X 0,Y 587.198,Z 359.236,A -85,B 0,C 180,E1 -1376.285,E2 -1376.285} C_VEL
LIN {X 0,Y 587.189,Z 354.596,A -85,B 0,C 180,E1 -1377.359,E2 -1377.359} C_VEL
LIN {X 0,Y 587.223,Z 348.81,A -85,B 0,C 180,E1 -1378.407,E2 -1378.407} C_VEL
LIN {X 0,Y 587.237,Z 342.091,A -85,B 0,C 180,E1 -1379.386,E2 -1379.386} C_VEL
LIN {X 0,Y 587.297,Z 334.065,A -85,B 0,C 180,E1 -1380.338,E2 -1380.338} C_VEL
LIN {X 0,Y 587.379,Z 324.511,A -85,B 0,C 180,E1 -1381.264,E2 -1381.264} C_VEL
LIN {X 0,Y 587.407,Z 314.173,A -85,B 0,C 180,E1 -1382.075,E2 -1382.075} C_VEL
LIN {X 0,Y 587.488,Z 303.36,A -85,B 0,C 180,E1 -1382.754,E2 -1382.754} C_VEL
LIN {X 0,Y 587.582,Z 292.338,A -85,B 0,C 180,E1 -1383.303,E2 -1383.303} C_VEL
LIN {X 0,Y 587.653,Z 279.523,A -85,B 0,C 180,E1 -1383.787,E2 -1383.787} C_VEL
LIN {X 0,Y 587.692,Z 266.598,A -85,B 0,C 180,E1 -1384.121,E2 -1384.121} C_VEL
LIN {X 0,Y 587.719,Z 248.198,A -85,B 0,C 180,E1 -1384.387,E2 -1384.387} C_VEL
LIN {X 0,Y 587.708,Z 158.623,A -85,B 0,C 180,E1 -1385.487,E2 -1385.487} C_VEL
LIN {X 0,Y 587.341,Z 156.327,A -85,B 0,C 180,E1 -1385.54,E2 -1385.54} C_VEL
LIN {X 0,Y 587.425,Z 141.529,A -85,B 0,C 180,E1 -1388.126,E2 -1388.126} C_VEL
LIN {X 0,Y 587.48,Z 126.112,A -85,B 0,C 180,E1 -1390.858,E2 -1390.858} C_VEL
LIN {X 0,Y 587.342,Z 125.322,A -85,B 0,C 180,E1 -1391.02,E2 -1391.02} C_VEL
LIN {X 0,Y 587.332,Z 125.329,A -85,B 0,C 180,E1 -1393.95,E2 -1393.95} C_VEL
LIN {X 0,Y 587.319,Z 125.321,A -85,B 0,C 180,E1 -1396.995,E2 -1396.995} C_VEL
LIN {X 0,Y 587.317,Z 125.331,A -85,B 0,C 180,E1 -1399.747,E2 -1399.747} C_VEL
LIN {X 0,Y 587.344,Z 125.319,A -85,B 0,C 180,E1 -1402.393,E2 -1402.393} C_VEL
LIN {X 0,Y 587.36,Z 125.323,A -85,B 0,C 180,E1 -1405.781,E2 -1405.781} C_VEL
LIN {X 0,Y 587.341,Z 125.319,A -85,B 0,C 180,E1 -1408.232,E2 -1408.232} C_VEL
LIN {X 0,Y 587.348,Z 125.319,A -85,B 0,C 180,E1 -1410.867,E2 -1410.867} C_VEL
LIN {X 0,Y 587.356,Z 125.319,A -85,B 0,C 180,E1 -1413.82,E2 -1413.82} C_VEL
LIN {X 0,Y 587.323,Z 125.321,A -85,B 0,C 180,E1 -1415.994,E2 -1415.994} C_VEL
LIN {X 0,Y 587.317,Z 125.321,A -85,B 0,C 180,E1 -1418.226,E2 -1418.226} C_VEL
LIN {X 0,Y 587.344,Z 125.326,A -85,B 0,C 180,E1 -1421.152,E2 -1421.152} C_VEL
LIN {X 0,Y 587.314,Z 125.321,A -85,B 0,C 180,E1 -1424.025,E2 -1424.025} C_VEL
LIN {X 0,Y 587.31,Z 125.331,A -85,B 0,C 180,E1 -1426.859,E2 -1426.859} C_VEL
LIN {X 0,Y 587.334,Z 125.319,A -85,B 0,C 180,E1 -1429.661,E2 -1429.661} C_VEL
LIN {X 0,Y 587.363,Z 125.32,A -85,B 0,C 180,E1 -1432.437,E2 -1432.437} C_VEL
LIN {X 0,Y 587.343,Z 125.318,A -85,B 0,C 180,E1 -1435.196,E2 -1435.196} C_VEL
LIN {X 0,Y 587.372,Z 125.315,A -85,B 0,C 180,E1 -1437.943,E2 -1437.943} C_VEL
LIN {X 0,Y 587.384,Z 125.317,A -85,B 0,C 180,E1 -1440.686,E2 -1440.686} C_VEL
LIN {X 0,Y 587.356,Z 125.319,A -85,B 0,C 180,E1 -1442.744,E2 -1442.744} C_VEL
LIN {X 0,Y 587.342,Z 125.317,A -85,B 0,C 180,E1 -1445.494,E2 -1445.494} C_VEL
LIN {X 0,Y 587.339,Z 125.326,A -85,B 0,C 180,E1 -1448.256,E2 -1448.256} C_VEL
LIN {X 0,Y 587.334,Z 125.317,A -85,B 0,C 180,E1 -1451.125,E2 -1451.125} C_VEL
LIN {X 0,Y 587.33,Z 125.324,A -85,B 0,C 180,E1 -1454.246,E2 -1454.246} C_VEL
LIN {X 0,Y 587.282,Z 125.324,A -85,B 0,C 180,E1 -1456.792,E2 -1456.792} C_VEL
LIN {X 0,Y 587.299,Z 125.33,A -85,B 0,C 180,E1 -1459.577,E2 -1459.577} C_VEL
LIN {X 0,Y 587.298,Z 125.332,A -85,B 0,C 180,E1 -1461.776,E2 -1461.776} C_VEL
LIN {X 0,Y 587.302,Z 125.323,A -85,B 0,C 180,E1 -1464.761,E2 -1464.761} C_VEL
LIN {X 0,Y 587.298,Z 125.33,A -85,B 0,C 180,E1 -1467.682,E2 -1467.682} C_VEL
LIN {X 0,Y 587.288,Z 125.324,A -85,B 0,C 180,E1 -1470.501,E2 -1470.501} C_VEL
LIN {X 0,Y 587.304,Z 125.331,A -85,B 0,C 180,E1 -1473.399,E2 -1473.399} C_VEL
LIN {X 0,Y 587.253,Z 125.33,A -85,B 0,C 180,E1 -1475.903,E2 -1475.903} C_VEL
LIN {X 0,Y 587.271,Z 125.327,A -85,B 0,C 180,E1 -1478.484,E2 -1478.484} C_VEL
LIN {X 0,Y 587.298,Z 125.332,A -85,B 0,C 180,E1 -1481.161,E2 -1481.161} C_VEL
LIN {X 0,Y 587.304,Z 125.323,A -85,B 0,C 180,E1 -1484.111,E2 -1484.111} C_VEL
LIN {X 0,Y 587.283,Z 125.333,A -85,B 0,C 180,E1 -1486.991,E2 -1486.991} C_VEL
LIN {X 0,Y 587.293,Z 125.324,A -85,B 0,C 180,E1 -1489.744,E2 -1489.744} C_VEL
LIN {X 0,Y 587.332,Z 125.325,A -85,B 0,C 180,E1 -1492.391,E2 -1492.391} C_VEL
LIN {X 0,Y 587.328,Z 125.32,A -85,B 0,C 180,E1 -1495.656,E2 -1495.656} C_VEL
LIN {X 0,Y 587.334,Z 125.325,A -85,B 0,C 180,E1 -1498.231,E2 -1498.231} C_VEL
LIN {X 0,Y 587.341,Z 125.321,A -85,B 0,C 180,E1 -1500.869,E2 -1500.869} C_VEL
LIN {X 0,Y 587.31,Z 125.326,A -85,B 0,C 180,E1 -1503.83,E2 -1503.83} C_VEL
LIN {X 0,Y 587.315,Z 125.381,A -85,B 0,C 180,E1 -1506.847,E2 -1506.847} C_VEL
LIN {X 0,Y 587.834,Z 129.942,A -85,B 0,C 180,E1 -1507.506,E2 -1507.506} C_VEL
LIN {X 0,Y 587.74,Z 149.468,A -85,B 0,C 180,E1 -1510.257,E2 -1510.257} C_VEL
LIN {X 0,Y 587.525,Z 170.13,A -85,B 0,C 180,E1 -1513.13,E2 -1513.13} C_VEL
LIN {X 0,Y 587.451,Z 189.888,A -85,B 0,C 180,E1 -1515.843,E2 -1515.843} C_VEL
LIN {X 0,Y 587.381,Z 194.613,A -85,B 0,C 180,E1 -1516.486,E2 -1516.486} C_VEL
LIN {X 0,Y 587.838,Z 198.724,A -85,B 0,C 180,E1 -1516.562,E2 -1516.562} C_VEL
LIN {X 0,Y 587.724,Z 302.95,A -85,B 0,C 180,E1 -1517.855,E2 -1517.855} C_VEL
LIN {X 0,Y 587.668,Z 316.222,A -85,B 0,C 180,E1 -1518.16,E2 -1518.16} C_VEL
LIN {X 0,Y 587.606,Z 328.643,A -85,B 0,C 180,E1 -1518.585,E2 -1518.585} C_VEL
LIN {X 0,Y 587.557,Z 340.631,A -85,B 0,C 180,E1 -1519.141,E2 -1519.141} C_VEL
LIN {X 0,Y 587.464,Z 352.204,A -85,B 0,C 180,E1 -1519.837,E2 -1519.837} C_VEL
LIN {X 0,Y 587.366,Z 362.6,A -85,B 0,C 180,E1 -1520.617,E2 -1520.617} C_VEL
LIN {X 0,Y 587.322,Z 371.113,A -85,B 0,C 180,E1 -1521.398,E2 -1521.398} C_VEL
LIN {X 0,Y 587.274,Z 378.961,A -85,B 0,C 180,E1 -1522.263,E2 -1522.263} C_VEL
LIN {X 0,Y 587.23,Z 385.47,A -85,B 0,C 180,E1 -1523.126,E2 -1523.126} C_VEL
LIN {X 0,Y 587.237,Z 391.867,A -85,B 0,C 180,E1 -1524.161,E2 -1524.161} C_VEL
LIN {X 0,Y 587.147,Z 396.95,A -85,B 0,C 180,E1 -1525.194,E2 -1525.194} C_VEL
LIN {X 0,Y 587.213,Z 400.896,A -85,B 0,C 180,E1 -1526.226,E2 -1526.226} C_VEL
LIN {X 0,Y 587.132,Z 403.809,A -85,B 0,C 180,E1 -1527.256,E2 -1527.256} C_VEL
LIN {X 0,Y 587.141,Z 405.2,A -85,B 0,C 180,E1 -1527.942,E2 -1527.942} C_VEL
LIN {X 0,Y 587.14,Z 406.785,A -85,B 0,C 180,E1 -1529.314,E2 -1529.314} C_VEL
LIN {X 0,Y 587.137,Z 407,A -85,B 0,C 180,E1 -1530,E2 -1530} C_VEL
LIN {X 0,Y 587.147,Z 406.186,A -85,B 0,C 180,E1 -1531.372,E2 -1531.372} C_VEL
LIN {X 0,Y 587.141,Z 405.2,A -85,B 0,C 180,E1 -1532.058,E2 -1532.058} C_VEL
LIN {X 0,Y 587.132,Z 403.809,A -85,B 0,C 180,E1 -1532.745,E2 -1532.745} C_VEL
LIN {X 0,Y 587.213,Z 400.895,A -85,B 0,C 180,E1 -1533.774,E2 -1533.774} C_VEL
LIN {X 0,Y 587.147,Z 396.948,A -85,B 0,C 180,E1 -1534.807,E2 -1534.807} C_VEL
LIN {X 0,Y 587.218,Z 390.876,A -85,B 0,C 180,E1 -1536.011,E2 -1536.011} C_VEL
LIN {X 0,Y 587.245,Z 384.236,A -85,B 0,C 180,E1 -1537.046,E2 -1537.046} C_VEL
LIN {X 0,Y 587.3,Z 375.989,A -85,B 0,C 180,E1 -1538.083,E2 -1538.083} C_VEL
LIN {X 0,Y 587.343,Z 367.536,A -85,B 0,C 180,E1 -1538.949,E2 -1538.949} C_VEL
LIN {X 0,Y 587.419,Z 357.094,A -85,B 0,C 180,E1 -1539.817,E2 -1539.817} C_VEL
LIN {X 0,Y 587.497,Z 346.753,A -85,B 0,C 180,E1 -1540.512,E2 -1540.512} C_VEL
LIN {X 0,Y 587.561,Z 334.815,A -85,B 0,C 180,E1 -1541.149,E2 -1541.149} C_VEL
LIN {X 0,Y 587.63,Z 322.593,A -85,B 0,C 180,E1 -1541.639,E2 -1541.639} C_VEL
LIN {X 0,Y 587.704,Z 309.425,A -85,B 0,C 180,E1 -1542.014,E2 -1542.014} C_VEL
LIN {X 0,Y 587.785,Z 297.067,A -85,B 0,C 180,E1 -1542.232,E2 -1542.232} C_VEL
LIN {X 0,Y 587.709,Z 196.688,A -85,B 0,C 180,E1 -1543.466,E2 -1543.466} C_VEL
LIN {X 0,Y 587.381,Z 194.611,A -85,B 0,C 180,E1 -1543.515,E2 -1543.515} C_VEL
LIN {X 0,Y 587.542,Z 174.061,A -85,B 0,C 180,E1 -1546.326,E2 -1546.326} C_VEL
LIN {X 0,Y 587.67,Z 153.849,A -85,B 0,C 180,E1 -1549.131,E2 -1549.131} C_VEL
LIN {X 0,Y 587.806,Z 133.908,A -85,B 0,C 180,E1 -1551.94,E2 -1551.94} C_VEL
LIN {X 0,Y 587.61,Z 126.884,A -85,B 0,C 180,E1 -1552.935,E2 -1552.935} C_VEL
LIN {X 0,Y 587.315,Z 125.326,A -85,B 0,C 180,E1 -1553.18,E2 -1553.18} C_VEL
LIN {X 0,Y 587.311,Z 125.326,A -85,B 0,C 180,E1 -1556.171,E2 -1556.171} C_VEL
LIN {X 0,Y 587.344,Z 125.319,A -85,B 0,C 180,E1 -1559.132,E2 -1559.132} C_VEL
LIN {X 0,Y 587.318,Z 125.327,A -85,B 0,C 180,E1 -1561.831,E2 -1561.831} C_VEL
LIN {X 0,Y 587.332,Z 125.319,A -85,B 0,C 180,E1 -1564.345,E2 -1564.345} C_VEL
LIN {X 0,Y 587.341,Z 125.326,A -85,B 0,C 180,E1 -1567.608,E2 -1567.608} C_VEL
LIN {X 0,Y 587.298,Z 125.323,A -85,B 0,C 180,E1 -1570.256,E2 -1570.256} C_VEL
LIN {X 0,Y 587.293,Z 125.33,A -85,B 0,C 180,E1 -1573.115,E2 -1573.115} C_VEL
LIN {X 0,Y 587.302,Z 125.323,A -85,B 0,C 180,E1 -1576.047,E2 -1576.047} C_VEL
LIN {X 0,Y 587.335,Z 125.324,A -85,B 0,C 180,E1 -1578.926,E2 -1578.926} C_VEL
LIN {X 0,Y 587.316,Z 125.325,A -85,B 0,C 180,E1 -1581.519,E2 -1581.519} C_VEL
LIN {X 0,Y 587.28,Z 125.325,A -85,B 0,C 180,E1 -1584.099,E2 -1584.099} C_VEL
LIN {X 0,Y 587.336,Z 125.326,A -85,B 0,C 180,E1 -1586.89,E2 -1586.89} C_VEL
LIN {X 0,Y 587.298,Z 125.323,A -85,B 0,C 180,E1 -1589.827,E2 -1589.827} C_VEL
LIN {X 0,Y 587.302,Z 125.324,A -85,B 0,C 180,E1 -1592.317,E2 -1592.317} C_VEL
LIN {X 0,Y 587.302,Z 125.326,A -85,B 0,C 180,E1 -1595.239,E2 -1595.239} C_VEL
LIN {X 0,Y 587.302,Z 125.325,A -85,B 0,C 180,E1 -1598.224,E2 -1598.224} C_VEL
LIN {X 0,Y 587.327,Z 125.322,A -85,B 0,C 180,E1 -1601.15,E2 -1601.15} C_VEL
LIN {X 0,Y 587.291,Z 125.325,A -85,B 0,C 180,E1 -1604.023,E2 -1604.023} C_VEL
LIN {X 0,Y 587.328,Z 125.323,A -85,B 0,C 180,E1 -1606.153,E2 -1606.153} C_VEL
LIN {X 0,Y 587.344,Z 125.32,A -85,B 0,C 180,E1 -1608.962,E2 -1608.962} C_VEL
LIN {X 0,Y 587.33,Z 125.32,A -85,B 0,C 180,E1 -1611.744,E2 -1611.744} C_VEL
LIN {X 0,Y 587.34,Z 125.325,A -85,B 0,C 180,E1 -1614.506,E2 -1614.506} C_VEL
LIN {X 0,Y 587.338,Z 125.318,A -85,B 0,C 180,E1 -1617.256,E2 -1617.256} C_VEL
LIN {X 0,Y 587.383,Z 125.319,A -85,B 0,C 180,E1 -1619.999,E2 -1619.999} C_VEL
LIN {X 0,Y 587.342,Z 125.319,A -85,B 0,C 180,E1 -1622.743,E2 -1622.743} C_VEL
LIN {X 0,Y 587.331,Z 125.32,A -85,B 0,C 180,E1 -1625.493,E2 -1625.493} C_VEL
LIN {X 0,Y 587.332,Z 125.325,A -85,B 0,C 180,E1 -1628.255,E2 -1628.255} C_VEL
LIN {X 0,Y 587.319,Z 125.32,A -85,B 0,C 180,E1 -1631.116,E2 -1631.116} C_VEL
LIN {X 0,Y 587.344,Z 125.327,A -85,B 0,C 180,E1 -1633.845,E2 -1633.845} C_VEL
LIN {X 0,Y 587.278,Z 125.325,A -85,B 0,C 180,E1 -1636.789,E2 -1636.789} C_VEL
LIN {X 0,Y 587.278,Z 125.328,A -85,B 0,C 180,E1 -1638.272,E2 -1638.272} C_VEL
LIN {X 0,Y 586.624,Z 125.409,A -85,B 0,C 180,E1 -1638.844,E2 -1638.844} C_VEL
LIN {X 0,Y 583.768,Z 125.773,A -85,B 0,C 180,E1 -1639.772,E2 -1639.772} C_VEL
LIN {X 0,Y 581.359,Z 126.067,A -85,B 0,C 180,E1 -1640.519,E2 -1640.519} C_VEL
LIN {X 0,Y 580.34,Z 126.191,A -85,B 0,C 180,E1 -1641.096,E2 -1641.096} C_VEL
LIN {X 0,Y 580.267,Z 126.202,A -85,B 0,C 180,E1 -1641.291,E2 -1641.291} C_VEL
LIN {X 0,Y 580.249,Z 126.202,A -85,B 0,C 180,E1 -1644.318,E2 -1644.318} C_VEL
LIN {X 0,Y 580.241,Z 126.202,A -85,B 0,C 180,E1 -1646.624,E2 -1646.624} C_VEL
LIN {X 0,Y 580.249,Z 126.207,A -85,B 0,C 180,E1 -1649.299,E2 -1649.299} C_VEL
LIN {X 0,Y 580.281,Z 126.198,A -85,B 0,C 180,E1 -1652.201,E2 -1652.201} C_VEL
LIN {X 0,Y 580.271,Z 126.199,A -85,B 0,C 180,E1 -1654.697,E2 -1654.697} C_VEL
LIN {X 0,Y 580.28,Z 126.206,A -85,B 0,C 180,E1 -1657.269,E2 -1657.269} C_VEL
LIN {X 0,Y 580.27,Z 126.198,A -85,B 0,C 180,E1 -1660.267,E2 -1660.267} C_VEL
LIN {X 0,Y 580.23,Z 126.21,A -85,B 0,C 180,E1 -1663.385,E2 -1663.385} C_VEL
LIN {X 0,Y 580.232,Z 126.204,A -85,B 0,C 180,E1 -1666.337,E2 -1666.337} C_VEL
LIN {X 0,Y 580.271,Z 126.206,A -85,B 0,C 180,E1 -1669.154,E2 -1669.154} C_VEL
LIN {X 0,Y 580.276,Z 126.198,A -85,B 0,C 180,E1 -1671.928,E2 -1671.928} C_VEL
LIN {X 0,Y 580.218,Z 126.208,A -85,B 0,C 180,E1 -1674.45,E2 -1674.45} C_VEL
LIN {X 0,Y 580.275,Z 126.206,A -85,B 0,C 180,E1 -1676.974,E2 -1676.974} C_VEL
LIN {X 0,Y 580.261,Z 126.201,A -85,B 0,C 180,E1 -1679.423,E2 -1679.423} C_VEL
LIN {X 0,Y 580.234,Z 126.205,A -85,B 0,C 180,E1 -1682.152,E2 -1682.152} C_VEL
LIN {X 0,Y 580.269,Z 126.204,A -85,B 0,C 180,E1 -1684.918,E2 -1684.918} C_VEL
LIN {X 0,Y 580.223,Z 126.205,A -85,B 0,C 180,E1 -1687.945,E2 -1687.945} C_VEL
LIN {X 0,Y 580.269,Z 126.202,A -85,B 0,C 180,E1 -1690.912,E2 -1690.912} C_VEL
LIN {X 0,Y 580.226,Z 126.205,A -85,B 0,C 180,E1 -1693.824,E2 -1693.824} C_VEL
LIN {X 0,Y 580.284,Z 126.2,A -85,B 0,C 180,E1 -1695.982,E2 -1695.982} C_VEL
LIN {X 0,Y 580.259,Z 126.202,A -85,B 0,C 180,E1 -1698.826,E2 -1698.826} C_VEL
LIN {X 0,Y 580.286,Z 126.198,A -85,B 0,C 180,E1 -1701.643,E2 -1701.643} C_VEL
LIN {X 0,Y 580.294,Z 126.201,A -85,B 0,C 180,E1 -1704.44,E2 -1704.44} C_VEL
LIN {X 0,Y 580.334,Z 126.198,A -85,B 0,C 180,E1 -1707.918,E2 -1707.918} C_VEL
LIN {X 0,Y 580.341,Z 126.2,A -85,B 0,C 180,E1 -1710,E2 -1710} C_VEL
LIN {X 0,Y 580.29,Z 126.2,A -85,B 0,C 180,E1 -1712.777,E2 -1712.777} C_VEL
LIN {X 0,Y 580.269,Z 126.372,A -85,B 0,C 180,E1 -1713.037,E2 -1713.037} C_VEL
LIN {X 0,Y 580.344,Z 136.497,A -85,B 0,C 180,E1 -1714.863,E2 -1714.863} C_VEL
LIN {X 0,Y 580.32,Z 150.22,A -85,B 0,C 180,E1 -1717.305,E2 -1717.305} C_VEL
LIN {X 0,Y 580.282,Z 156.437,A -85,B 0,C 180,E1 -1718.4,E2 -1718.4} C_VEL
LIN {X 0,Y 580.956,Z 161.385,A -85,B 0,C 180,E1 -1718.478,E2 -1718.478} C_VEL
LIN {X 0,Y 580.776,Z 263.007,A -85,B 0,C 180,E1 -1719.754,E2 -1719.754} C_VEL
LIN {X 0,Y 580.677,Z 276.304,A -85,B 0,C 180,E1 -1720.063,E2 -1720.063} C_VEL
LIN {X 0,Y 580.629,Z 288.982,A -85,B 0,C 180,E1 -1720.505,E2 -1720.505} C_VEL
LIN {X 0,Y 580.56,Z 301.096,A -85,B 0,C 180,E1 -1721.08,E2 -1721.08} C_VEL
LIN {X 0,Y 580.433,Z 312.682,A -85,B 0,C 180,E1 -1721.79,E2 -1721.79} C_VEL
LIN {X 0,Y 580.375,Z 323.1,A -85,B 0,C 180,E1 -1722.59,E2 -1722.59} C_VEL
LIN {X 0,Y 580.292,Z 332.498,A -85,B 0,C 180,E1 -1723.482,E2 -1723.482} C_VEL
LIN {X 0,Y 580.222,Z 340.923,A -85,B 0,C 180,E1 -1724.464,E2 -1724.464} C_VEL
LIN {X 0,Y 580.161,Z 347.865,A -85,B 0,C 180,E1 -1725.456,E2 -1725.456} C_VEL
LIN {X 0,Y 580.099,Z 353.854,A -85,B 0,C 180,E1 -1726.517,E2 -1726.517} C_VEL
LIN {X 0,Y 580.091,Z 358.788,A -85,B 0,C 180,E1 -1727.631,E2 -1727.631} C_VEL
LIN {X 0,Y 580.064,Z 362.413,A -85,B 0,C 180,E1 -1728.723,E2 -1728.723} C_VEL
LIN {X 0,Y 580.046,Z 364.983,A -85,B 0,C 180,E1 -1729.831,E2 -1729.831} C_VEL
LIN {X 0,Y 580.058,Z 366.619,A -85,B 0,C 180,E1 -1731.105,E2 -1731.105} C_VEL
LIN {X 0,Y 580.028,Z 366.999,A -85,B 0,C 180,E1 -1732.062,E2 -1732.062} C_VEL
LIN {X 0,Y 580.041,Z 366.641,A -85,B 0,C 180,E1 -1732.952,E2 -1732.952} C_VEL
LIN {X 0,Y 580.025,Z 364.843,A -85,B 0,C 180,E1 -1734.329,E2 -1734.329} C_VEL
LIN {X 0,Y 580.072,Z 362.09,A -85,B 0,C 180,E1 -1735.474,E2 -1735.474} C_VEL
LIN {X 0,Y 580.112,Z 358.086,A -85,B 0,C 180,E1 -1736.632,E2 -1736.632} C_VEL
LIN {X 0,Y 580.117,Z 352.539,A -85,B 0,C 180,E1 -1737.827,E2 -1737.827} C_VEL
LIN {X 0,Y 580.157,Z 345.603,A -85,B 0,C 180,E1 -1738.984,E2 -1738.984} C_VEL
LIN {X 0,Y 580.221,Z 338.118,A -85,B 0,C 180,E1 -1739.977,E2 -1739.977} C_VEL
LIN {X 0,Y 580.308,Z 328.546,A -85,B 0,C 180,E1 -1741.006,E2 -1741.006} C_VEL
LIN {X 0,Y 580.37,Z 318.402,A -85,B 0,C 180,E1 -1741.883,E2 -1741.883} C_VEL
LIN {X 0,Y 580.468,Z 308.112,A -85,B 0,C 180,E1 -1742.601,E2 -1742.601} C_VEL
LIN {X 0,Y 580.577,Z 295.638,A -85,B 0,C 180,E1 -1743.29,E2 -1743.29} C_VEL
LIN {X 0,Y 580.671,Z 283.545,A -85,B 0,C 180,E1 -1743.794,E2 -1743.794} C_VEL
LIN {X 0,Y 580.757,Z 269.988,A -85,B 0,C 180,E1 -1744.192,E2 -1744.192} C_VEL
LIN {X 0,Y 580.81,Z 257.186,A -85,B 0,C 180,E1 -1744.424,E2 -1744.424} C_VEL
LIN {X 0,Y 580.909,Z 160.094,A -85,B 0,C 180,E1 -1745.629,E2 -1745.629} C_VEL
LIN {X 0,Y 580.301,Z 156.341,A -85,B 0,C 180,E1 -1745.704,E2 -1745.704} C_VEL
LIN {X 0,Y 580.395,Z 141.346,A -85,B 0,C 180,E1 -1748.359,E2 -1748.359} C_VEL
LIN {X 0,Y 580.492,Z 127.581,A -85,B 0,C 180,E1 -1750.827,E2 -1750.827} C_VEL
LIN {X 0,Y 580.32,Z 126.197,A -85,B 0,C 180,E1 -1751.086,E2 -1751.086} C_VEL
LIN {X 0,Y 580.285,Z 126.203,A -85,B 0,C 180,E1 -1753.657,E2 -1753.657} C_VEL
LIN {X 0,Y 580.283,Z 126.198,A -85,B 0,C 180,E1 -1756.609,E2 -1756.609} C_VEL
LIN {X 0,Y 580.298,Z 126.197,A -85,B 0,C 180,E1 -1759.158,E2 -1759.158} C_VEL
LIN {X 0,Y 580.289,Z 126.204,A -85,B 0,C 180,E1 -1761.927,E2 -1761.927} C_VEL
LIN {X 0,Y 580.249,Z 126.202,A -85,B 0,C 180,E1 -1764.453,E2 -1764.453} C_VEL
LIN {X 0,Y 580.29,Z 126.198,A -85,B 0,C 180,E1 -1766.976,E2 -1766.976} C_VEL
LIN {X 0,Y 580.294,Z 126.205,A -85,B 0,C 180,E1 -1769.426,E2 -1769.426} C_VEL
LIN {X 0,Y 580.297,Z 126.196,A -85,B 0,C 180,E1 -1772.142,E2 -1772.142} C_VEL
LIN {X 0,Y 580.321,Z 126.202,A -85,B 0,C 180,E1 -1775.271,E2 -1775.271} C_VEL
LIN {X 0,Y 580.269,Z 126.2,A -85,B 0,C 180,E1 -1777.948,E2 -1777.948} C_VEL
LIN {X 0,Y 580.296,Z 126.203,A -85,B 0,C 180,E1 -1780.914,E2 -1780.914} C_VEL
LIN {X 0,Y 580.264,Z 126.2,A -85,B 0,C 180,E1 -1783.826,E2 -1783.826} C_VEL
LIN {X 0,Y 580.267,Z 126.205,A -85,B 0,C 180,E1 -1786.696,E2 -1786.696} C_VEL
LIN {X 0,Y 580.307,Z 126.204,A -85,B 0,C 180,E1 -1788.828,E2 -1788.828} C_VEL
LIN {X 0,Y 580.309,Z 126.193,A -85,B 0,C 180,E1 -1791.644,E2 -1791.644} C_VEL
LIN {X 0,Y 580.329,Z 126.198,A -85,B 0,C 180,E1 -1794.441,E2 -1794.441} C_VEL
LIN {X 0,Y 580.342,Z 126.191,A -85,B 0,C 180,E1 -1797.919,E2 -1797.919} C_VEL
LIN {X 0,Y 580.355,Z 126.192,A -85,B 0,C 180,E1 -1800.694,E2 -1800.694} C_VEL
LIN {X 0,Y 580.322,Z 126.195,A -85,B 0,C 180,E1 -1802.777,E2 -1802.777} C_VEL
LIN {X 0,Y 580.312,Z 126.193,A -85,B 0,C 180,E1 -1805.56,E2 -1805.56} C_VEL
LIN {X 0,Y 580.307,Z 126.2,A -85,B 0,C 180,E1 -1808.357,E2 -1808.357} C_VEL
LIN {X 0,Y 580.305,Z 126.193,A -85,B 0,C 180,E1 -1811.191,E2 -1811.191} C_VEL
LIN {X 0,Y 580.291,Z 126.2,A -85,B 0,C 180,E1 -1814.328,E2 -1814.328} C_VEL
LIN {X 0,Y 580.232,Z 126.202,A -85,B 0,C 180,E1 -1816.9,E2 -1816.9} C_VEL
LIN {X 0,Y 580.273,Z 126.207,A -85,B 0,C 180,E1 -1819.824,E2 -1819.824} C_VEL
LIN {X 0,Y 580.232,Z 126.207,A -85,B 0,C 180,E1 -1822.055,E2 -1822.055} C_VEL
LIN {X 0,Y 580.281,Z 126.2,A -85,B 0,C 180,E1 -1825.081,E2 -1825.081} C_VEL
LIN {X 0,Y 580.24,Z 126.207,A -85,B 0,C 180,E1 -1827.847,E2 -1827.847} C_VEL
LIN {X 0,Y 580.241,Z 126.202,A -85,B 0,C 180,E1 -1830.687,E2 -1830.687} C_VEL
LIN {X 0,Y 580.252,Z 126.211,A -85,B 0,C 180,E1 -1833.308,E2 -1833.308} C_VEL
LIN {X 0,Y 580.203,Z 126.209,A -85,B 0,C 180,E1 -1835.75,E2 -1835.75} C_VEL
LIN {X 0,Y 580.235,Z 126.203,A -85,B 0,C 180,E1 -1838.151,E2 -1838.151} C_VEL
LIN {X 0,Y 580.249,Z 126.208,A -85,B 0,C 180,E1 -1840.848,E2 -1840.848} C_VEL
LIN {X 0,Y 580.235,Z 126.204,A -85,B 0,C 180,E1 -1843.662,E2 -1843.662} C_VEL
LIN {X 0,Y 580.236,Z 126.206,A -85,B 0,C 180,E1 -1846.338,E2 -1846.338} C_VEL
LIN {X 0,Y 580.256,Z 126.205,A -85,B 0,C 180,E1 -1849.153,E2 -1849.153} C_VEL
LIN {X 0,Y 580.277,Z 126.199,A -85,B 0,C 180,E1 -1851.929,E2 -1851.929} C_VEL
LIN {X 0,Y 580.225,Z 126.211,A -85,B 0,C 180,E1 -1854.451,E2 -1854.451} C_VEL
LIN {X 0,Y 580.284,Z 126.2,A -85,B 0,C 180,E1 -1856.975,E2 -1856.975} C_VEL
LIN {X 0,Y 580.279,Z 126.198,A -85,B 0,C 180,E1 -1859.424,E2 -1859.424} C_VEL
LIN {X 0,Y 580.244,Z 126.209,A -85,B 0,C 180,E1 -1862.152,E2 -1862.152} C_VEL
LIN {X 0,Y 580.284,Z 126.2,A -85,B 0,C 180,E1 -1864.919,E2 -1864.919} C_VEL
LIN {X 0,Y 580.293,Z 126.388,A -85,B 0,C 180,E1 -1866.736,E2 -1866.736} C_VEL
LIN {X 0,Y 580.899,Z 130.976,A -85,B 0,C 180,E1 -1867.41,E2 -1867.41} C_VEL
LIN {X 0,Y 580.779,Z 151.921,A -85,B 0,C 180,E1 -1870.359,E2 -1870.359} C_VEL
LIN {X 0,Y 580.562,Z 174.063,A -85,B 0,C 180,E1 -1873.472,E2 -1873.472} C_VEL
LIN {X 0,Y 580.384,Z 194.613,A -85,B 0,C 180,E1 -1876.32,E2 -1876.32} C_VEL
LIN {X 0,Y 580.926,Z 200.513,A -85,B 0,C 180,E1 -1876.422,E2 -1876.422} C_VEL
LIN {X 0,Y 580.806,Z 302.95,A -85,B 0,C 180,E1 -1877.708,E2 -1877.708} C_VEL
LIN {X 0,Y 580.727,Z 316.221,A -85,B 0,C 180,E1 -1878.017,E2 -1878.017} C_VEL
LIN {X 0,Y 580.648,Z 328.377,A -85,B 0,C 180,E1 -1878.436,E2 -1878.436} C_VEL
LIN {X 0,Y 580.579,Z 340.629,A -85,B 0,C 180,E1 -1879.009,E2 -1879.009} C_VEL
LIN {X 0,Y 580.441,Z 352.202,A -85,B 0,C 180,E1 -1879.712,E2 -1879.712} C_VEL
LIN {X 0,Y 580.345,Z 362.602,A -85,B 0,C 180,E1 -1880.503,E2 -1880.503} C_VEL
LIN {X 0,Y 580.271,Z 371.113,A -85,B 0,C 180,E1 -1881.292,E2 -1881.292} C_VEL
LIN {X 0,Y 580.222,Z 378.961,A -85,B 0,C 180,E1 -1882.168,E2 -1882.168} C_VEL
LIN {X 0,Y 580.154,Z 386.652,A -85,B 0,C 180,E1 -1883.222,E2 -1883.222} C_VEL
LIN {X 0,Y 580.139,Z 393.681,A -85,B 0,C 180,E1 -1884.439,E2 -1884.439} C_VEL
LIN {X 0,Y 580.108,Z 398.372,A -85,B 0,C 180,E1 -1885.484,E2 -1885.484} C_VEL
LIN {X 0,Y 580.123,Z 401.958,A -85,B 0,C 180,E1 -1886.527,E2 -1886.527} C_VEL
LIN {X 0,Y 580.043,Z 403.808,A -85,B 0,C 180,E1 -1887.222,E2 -1887.222} C_VEL
LIN {X 0,Y 580.04,Z 405.198,A -85,B 0,C 180,E1 -1887.917,E2 -1887.917} C_VEL
LIN {X 0,Y 580.04,Z 406.785,A -85,B 0,C 180,E1 -1889.306,E2 -1889.306} C_VEL
LIN {X 0,Y 580.037,Z 407,A -85,B 0,C 180,E1 -1890,E2 -1890} C_VEL
LIN {X 0,Y 580.047,Z 406.186,A -85,B 0,C 180,E1 -1891.389,E2 -1891.389} C_VEL
LIN {X 0,Y 580.04,Z 405.199,A -85,B 0,C 180,E1 -1892.083,E2 -1892.083} C_VEL
LIN {X 0,Y 580.043,Z 403.809,A -85,B 0,C 180,E1 -1892.778,E2 -1892.778} C_VEL
LIN {X 0,Y 580.11,Z 400.895,A -85,B 0,C 180,E1 -1893.821,E2 -1893.821} C_VEL
LIN {X 0,Y 580.053,Z 396.948,A -85,B 0,C 180,E1 -1894.865,E2 -1894.865} C_VEL
LIN {X 0,Y 580.139,Z 390.876,A -85,B 0,C 180,E1 -1896.085,E2 -1896.085} C_VEL
LIN {X 0,Y 580.185,Z 384.236,A -85,B 0,C 180,E1 -1897.133,E2 -1897.133} C_VEL
LIN {X 0,Y 580.25,Z 375.989,A -85,B 0,C 180,E1 -1898.182,E2 -1898.182} C_VEL
LIN {X 0,Y 580.308,Z 367.536,A -85,B 0,C 180,E1 -1899.059,E2 -1899.059} C_VEL
LIN {X 0,Y 580.422,Z 357.095,A -85,B 0,C 180,E1 -1899.936,E2 -1899.936} C_VEL
LIN {X 0,Y 580.506,Z 346.751,A -85,B 0,C 180,E1 -1900.64,E2 -1900.64} C_VEL
LIN {X 0,Y 580.597,Z 335.245,A -85,B 0,C 180,E1 -1901.264,E2 -1901.264} C_VEL
LIN {X 0,Y 580.683,Z 322.465,A -85,B 0,C 180,E1 -1901.785,E2 -1901.785} C_VEL
LIN {X 0,Y 580.778,Z 309.424,A -85,B 0,C 180,E1 -1902.16,E2 -1902.16} C_VEL
LIN {X 0,Y 580.869,Z 297.067,A -85,B 0,C 180,E1 -1902.379,E2 -1902.379} C_VEL
LIN {X 0,Y 580.793,Z 197.361,A -85,B 0,C 180,E1 -1903.621,E2 -1903.621} C_VEL
LIN {X 0,Y 580.387,Z 194.611,A -85,B 0,C 180,E1 -1903.681,E2 -1903.681} C_VEL
LIN {X 0,Y 580.565,Z 172.767,A -85,B 0,C 180,E1 -1906.709,E2 -1906.709} C_VEL
LIN {X 0,Y 580.783,Z 150.761,A -85,B 0,C 180,E1 -1909.806,E2 -1909.806} C_VEL
LIN {X 0,Y 580.899,Z 131.03,A -85,B 0,C 180,E1 -1912.59,E2 -1912.59} C_VEL
LIN {X 0,Y 580.262,Z 126.206,A -85,B 0,C 180,E1 -1913.339,E2 -1913.339} C_VEL
LIN {X 0,Y 580.265,Z 126.208,A -85,B 0,C 180,E1 -1915.851,E2 -1915.851} C_VEL
LIN {X 0,Y 580.282,Z 126.198,A -85,B 0,C 180,E1 -1918.977,E2 -1918.977} C_VEL
LIN {X 0,Y 580.27,Z 126.205,A -85,B 0,C 180,E1 -1921.386,E2 -1921.386} C_VEL
LIN {X 0,Y 580.277,Z 126.203,A -85,B 0,C 180,E1 -1923.858,E2 -1923.858} C_VEL
LIN {X 0,Y 580.28,Z 126.199,A -85,B 0,C 180,E1 -1926.931,E2 -1926.931} C_VEL
LIN {X 0,Y 580.274,Z 126.2,A -85,B 0,C 180,E1 -1929.935,E2 -1929.935} C_VEL
LIN {X 0,Y 580.255,Z 126.201,A -85,B 0,C 180,E1 -1932.709,E2 -1932.709} C_VEL
LIN {X 0,Y 580.255,Z 126.205,A -85,B 0,C 180,E1 -1935.611,E2 -1935.611} C_VEL
LIN {X 0,Y 580.273,Z 126.2,A -85,B 0,C 180,E1 -1938.67,E2 -1938.67} C_VEL
LIN {X 0,Y 580.268,Z 126.205,A -85,B 0,C 180,E1 -1940.964,E2 -1940.964} C_VEL
LIN {X 0,Y 580.248,Z 126.204,A -85,B 0,C 180,E1 -1943.594,E2 -1943.594} C_VEL
LIN {X 0,Y 580.277,Z 126.198,A -85,B 0,C 180,E1 -1946.142,E2 -1946.142} C_VEL
LIN {X 0,Y 580.257,Z 126.204,A -85,B 0,C 180,E1 -1948.613,E2 -1948.613} C_VEL
LIN {X 0,Y 580.281,Z 126.205,A -85,B 0,C 180,E1 -1951.023,E2 -1951.023} C_VEL
LIN {X 0,Y 580.268,Z 126.199,A -85,B 0,C 180,E1 -1953.672,E2 -1953.672} C_VEL
LIN {X 0,Y 580.247,Z 126.206,A -85,B 0,C 180,E1 -1956.44,E2 -1956.44} C_VEL
LIN {X 0,Y 580.256,Z 126.201,A -85,B 0,C 180,E1 -1959.436,E2 -1959.436} C_VEL
LIN {X 0,Y 580.24,Z 126.202,A -85,B 0,C 180,E1 -1961.644,E2 -1961.644} C_VEL
LIN {X 0,Y 580.271,Z 126.208,A -85,B 0,C 180,E1 -1964.546,E2 -1964.546} C_VEL
LIN {X 0,Y 580.27,Z 126.198,A -85,B 0,C 180,E1 -1967.407,E2 -1967.407} C_VEL
LIN {X 0,Y 580.291,Z 126.196,A -85,B 0,C 180,E1 -1969.533,E2 -1969.533} C_VEL
LIN {X 0,Y 580.294,Z 126.204,A -85,B 0,C 180,E1 -1972.344,E2 -1972.344} C_VEL
LIN {X 0,Y 580.303,Z 126.195,A -85,B 0,C 180,E1 -1975.136,E2 -1975.136} C_VEL
LIN {X 0,Y 580.34,Z 126.194,A -85,B 0,C 180,E1 -1977.917,E2 -1977.917} C_VEL
LIN {X 0,Y 580.263,Z 126.202,A -85,B 0,C 180,E1 -1980.693,E2 -1980.693} C_VEL
LIN {X 0,Y 580.31,Z 126.195,A -85,B 0,C 180,E1 -1982.776,E2 -1982.776} C_VEL
LIN {X 0,Y 580.3,Z 126.197,A -85,B 0,C 180,E1 -1985.559,E2 -1985.559} C_VEL
LIN {X 0,Y 580.298,Z 126.2,A -85,B 0,C 180,E1 -1988.356,E2 -1988.356} C_VEL
LIN {X 0,Y 580.271,Z 126.199,A -85,B 0,C 180,E1 -1991.173,E2 -1991.173} C_VEL
LIN {X 0,Y 580.303,Z 126.202,A -85,B 0,C 180,E1 -1994.017,E2 -1994.017} C_VEL
LIN {X 0,Y 580.228,Z 126.204,A -85,B 0,C 180,E1 -1996.899,E2 -1996.899} C_VEL
LIN {X 0,Y 580.271,Z 126.207,A -85,B 0,C 180,E1 -1999.823,E2 -1999.823} C_VEL
LIN {X 0,Y 580.267,Z 126.202,A -85,B 0,C 180,E1 -2001.291,E2 -2001.291} C_VEL
LIN {X 0,Y 579.617,Z 126.29,A -85,B 0,C 180,E1 -2001.871,E2 -2001.871} C_VEL
LIN {X 0,Y 576.738,Z 126.649,A -85,B 0,C 180,E1 -2002.81,E2 -2002.81} C_VEL
LIN {X 0,Y 574.301,Z 126.95,A -85,B 0,C 180,E1 -2003.566,E2 -2003.566} C_VEL
LIN {X 0,Y 573.27,Z 127.073,A -85,B 0,C 180,E1 -2004.15,E2 -2004.15} C_VEL
LIN {X 0,Y 573.195,Z 127.081,A -85,B 0,C 180,E1 -2004.348,E2 -2004.348} C_VEL
LIN {X 0,Y 573.188,Z 127.082,A -85,B 0,C 180,E1 -2006.978,E2 -2006.978} C_VEL
LIN {X 0,Y 573.199,Z 127.089,A -85,B 0,C 180,E1 -2009.479,E2 -2009.479} C_VEL
LIN {X 0,Y 573.235,Z 127.075,A -85,B 0,C 180,E1 -2012.225,E2 -2012.225} C_VEL
LIN {X 0,Y 573.217,Z 127.078,A -85,B 0,C 180,E1 -2014.768,E2 -2014.768} C_VEL
LIN {X 0,Y 573.218,Z 127.079,A -85,B 0,C 180,E1 -2017.808,E2 -2017.808} C_VEL
LIN {X 0,Y 573.225,Z 127.077,A -85,B 0,C 180,E1 -2020.526,E2 -2020.526} C_VEL
LIN {X 0,Y 573.196,Z 127.086,A -85,B 0,C 180,E1 -2023.362,E2 -2023.362} C_VEL
LIN {X 0,Y 573.201,Z 127.08,A -85,B 0,C 180,E1 -2026.335,E2 -2026.335} C_VEL
LIN {X 0,Y 573.241,Z 127.077,A -85,B 0,C 180,E1 -2029.474,E2 -2029.474} C_VEL
LIN {X 0,Y 573.22,Z 127.077,A -85,B 0,C 180,E1 -2032.191,E2 -2032.191} C_VEL
LIN {X 0,Y 573.212,Z 127.082,A -85,B 0,C 180,E1 -2035.231,E2 -2035.231} C_VEL
LIN {X 0,Y 573.23,Z 127.075,A -85,B 0,C 180,E1 -2037.774,E2 -2037.774} C_VEL
LIN {X 0,Y 573.224,Z 127.084,A -85,B 0,C 180,E1 -2040.632,E2 -2040.632} C_VEL
LIN {X 0,Y 573.199,Z 127.08,A -85,B 0,C 180,E1 -2043.513,E2 -2043.513} C_VEL
LIN {X 0,Y 573.185,Z 127.084,A -85,B 0,C 180,E1 -2046.132,E2 -2046.132} C_VEL
LIN {X 0,Y 573.218,Z 127.078,A -85,B 0,C 180,E1 -2049.172,E2 -2049.172} C_VEL
LIN {X 0,Y 573.185,Z 127.081,A -85,B 0,C 180,E1 -2051.41,E2 -2051.41} C_VEL
LIN {X 0,Y 573.195,Z 127.088,A -85,B 0,C 180,E1 -2054.351,E2 -2054.351} C_VEL
LIN {X 0,Y 573.187,Z 127.088,A -85,B 0,C 180,E1 -2056.528,E2 -2056.528} C_VEL
LIN {X 0,Y 573.231,Z 127.075,A -85,B 0,C 180,E1 -2059.403,E2 -2059.403} C_VEL
LIN {X 0,Y 573.211,Z 127.088,A -85,B 0,C 180,E1 -2062.249,E2 -2062.249} C_VEL
LIN {X 0,Y 573.266,Z 127.071,A -85,B 0,C 180,E1 -2065.077,E2 -2065.077} C_VEL
LIN {X 0,Y 573.303,Z 127.073,A -85,B 0,C 180,E1 -2067.892,E2 -2067.892} C_VEL
LIN {X 0,Y 573.309,Z 127.076,A -85,B 0,C 180,E1 -2070,E2 -2070} C_VEL
LIN {X 0,Y 573.253,Z 127.077,A -85,B 0,C 180,E1 -2072.811,E2 -2072.811} C_VEL
LIN {X 0,Y 573.255,Z 127.369,A -85,B 0,C 180,E1 -2072.987,E2 -2072.987} C_VEL
LIN {X 0,Y 573.357,Z 136.087,A -85,B 0,C 180,E1 -2074.57,E2 -2074.57} C_VEL
LIN {X 0,Y 573.274,Z 151.758,A -85,B 0,C 180,E1 -2077.396,E2 -2077.396} C_VEL
LIN {X 0,Y 573.256,Z 156.347,A -85,B 0,C 180,E1 -2078.216,E2 -2078.216} C_VEL
LIN {X 0,Y 574.039,Z 161.675,A -85,B 0,C 180,E1 -2078.315,E2 -2078.315} C_VEL
LIN {X 0,Y 573.856,Z 263.128,A -85,B 0,C 180,E1 -2079.606,E2 -2079.606} C_VEL
LIN {X 0,Y 573.729,Z 276.409,A -85,B 0,C 180,E1 -2079.919,E2 -2079.919} C_VEL
LIN {X 0,Y 573.665,Z 289.067,A -85,B 0,C 180,E1 -2080.366,E2 -2080.366} C_VEL
LIN {X 0,Y 573.587,Z 300.934,A -85,B 0,C 180,E1 -2080.936,E2 -2080.936} C_VEL
LIN {X 0,Y 573.41,Z 312.226,A -85,B 0,C 180,E1 -2081.632,E2 -2081.632} C_VEL
LIN {X 0,Y 573.343,Z 323.151,A -85,B 0,C 180,E1 -2082.477,E2 -2082.477} C_VEL
LIN {X 0,Y 573.235,Z 331.706,A -85,B 0,C 180,E1 -2083.29,E2 -2083.29} C_VEL
LIN {X 0,Y 573.146,Z 340.956,A -85,B 0,C 180,E1 -2084.374,E2 -2084.374} C_VEL
LIN {X 0,Y 573.081,Z 348.465,A -85,B 0,C 180,E1 -2085.47,E2 -2085.47} C_VEL
LIN {X 0,Y 573.034,Z 354.88,A -85,B 0,C 180,E1 -2086.661,E2 -2086.661} C_VEL
LIN {X 0,Y 572.993,Z 359.79,A -85,B 0,C 180,E1 -2087.857,E2 -2087.857} C_VEL
LIN {X 0,Y 572.96,Z 363.688,A -85,B 0,C 180,E1 -2089.183,E2 -2089.183} C_VEL
LIN {X 0,Y 572.97,Z 365.439,A -85,B 0,C 180,E1 -2090.087,E2 -2090.087} C_VEL
LIN {X 0,Y 572.973,Z 366.705,A -85,B 0,C 180,E1 -2091.221,E2 -2091.221} C_VEL
LIN {X 0,Y 572.933,Z 366.938,A -85,B 0,C 180,E1 -2092.35,E2 -2092.35} C_VEL
LIN {X 0,Y 572.931,Z 366.538,A -85,B 0,C 180,E1 -2093.112,E2 -2093.112} C_VEL
LIN {X 0,Y 572.923,Z 365.633,A -85,B 0,C 180,E1 -2093.879,E2 -2093.879} C_VEL
LIN {X 0,Y 572.953,Z 363.908,A -85,B 0,C 180,E1 -2094.812,E2 -2094.812} C_VEL
LIN {X 0,Y 572.999,Z 361.201,A -85,B 0,C 180,E1 -2095.812,E2 -2095.812} C_VEL
LIN {X 0,Y 573.003,Z 356.875,A -85,B 0,C 180,E1 -2096.989,E2 -2096.989} C_VEL
LIN {X 0,Y 573.049,Z 350.61,A -85,B 0,C 180,E1 -2098.252,E2 -2098.252} C_VEL
LIN {X 0,Y 573.091,Z 343.474,A -85,B 0,C 180,E1 -2099.376,E2 -2099.376} C_VEL
LIN {X 0,Y 573.174,Z 335.523,A -85,B 0,C 180,E1 -2100.384,E2 -2100.384} C_VEL
LIN {X 0,Y 573.285,Z 325.521,A -85,B 0,C 180,E1 -2101.4,E2 -2101.4} C_VEL
LIN {X 0,Y 573.381,Z 315.173,A -85,B 0,C 180,E1 -2102.25,E2 -2102.25} C_VEL
LIN {X 0,Y 573.506,Z 304.702,A -85,B 0,C 180,E1 -2102.942,E2 -2102.942} C_VEL
LIN {X 0,Y 573.638,Z 292.311,A -85,B 0,C 180,E1 -2103.582,E2 -2103.582} C_VEL
LIN {X 0,Y 573.766,Z 279.506,A -85,B 0,C 180,E1 -2104.076,E2 -2104.076} C_VEL
LIN {X 0,Y 573.839,Z 267.2,A -85,B 0,C 180,E1 -2104.405,E2 -2104.405} C_VEL
LIN {X 0,Y 573.867,Z 250.834,A -85,B 0,C 180,E1 -2104.656,E2 -2104.656} C_VEL
LIN {X 0,Y 574.005,Z 160.777,A -85,B 0,C 180,E1 -2105.787,E2 -2105.787} C_VEL
LIN {X 0,Y 573.267,Z 156.322,A -85,B 0,C 180,E1 -2105.878,E2 -2105.878} C_VEL
LIN {X 0,Y 573.402,Z 140.653,A -85,B 0,C 180,E1 -2108.689,E2 -2108.689} C_VEL
LIN {X 0,Y 573.406,Z 127.944,A -85,B 0,C 180,E1 -2110.974,E2 -2110.974} C_VEL
LIN {X 0,Y 573.291,Z 127.073,A -85,B 0,C 180,E1 -2111.159,E2 -2111.159} C_VEL
LIN {X 0,Y 573.236,Z 127.08,A -85,B 0,C 180,E1 -2114.334,E2 -2114.334} C_VEL
LIN {X 0,Y 573.241,Z 127.077,A -85,B 0,C 180,E1 -2117.359,E2 -2117.359} C_VEL
LIN {X 0,Y 573.245,Z 127.076,A -85,B 0,C 180,E1 -2120.394,E2 -2120.394} C_VEL
LIN {X 0,Y 573.25,Z 127.076,A -85,B 0,C 180,E1 -2123.078,E2 -2123.078} C_VEL
LIN {X 0,Y 573.266,Z 127.08,A -85,B 0,C 180,E1 -2125.672,E2 -2125.672} C_VEL
LIN {X 0,Y 573.24,Z 127.076,A -85,B 0,C 180,E1 -2128.185,E2 -2128.185} C_VEL
LIN {X 0,Y 573.263,Z 127.072,A -85,B 0,C 180,E1 -2130.635,E2 -2130.635} C_VEL
LIN {X 0,Y 573.25,Z 127.078,A -85,B 0,C 180,E1 -2133.025,E2 -2133.025} C_VEL
LIN {X 0,Y 573.273,Z 127.079,A -85,B 0,C 180,E1 -2135.367,E2 -2135.367} C_VEL
LIN {X 0,Y 573.228,Z 127.077,A -85,B 0,C 180,E1 -2138.42,E2 -2138.42} C_VEL
LIN {X 0,Y 573.269,Z 127.075,A -85,B 0,C 180,E1 -2140.732,E2 -2140.732} C_VEL
LIN {X 0,Y 573.24,Z 127.076,A -85,B 0,C 180,E1 -2143.622,E2 -2143.622} C_VEL
LIN {X 0,Y 573.224,Z 127.08,A -85,B 0,C 180,E1 -2146.53,E2 -2146.53} C_VEL
LIN {X 0,Y 573.265,Z 127.08,A -85,B 0,C 180,E1 -2148.746,E2 -2148.746} C_VEL
LIN {X 0,Y 573.253,Z 127.072,A -85,B 0,C 180,E1 -2151.541,E2 -2151.541} C_VEL
LIN {X 0,Y 573.295,Z 127.073,A -85,B 0,C 180,E1 -2154.372,E2 -2154.372} C_VEL
LIN {X 0,Y 573.312,Z 127.066,A -85,B 0,C 180,E1 -2157.893,E2 -2157.893} C_VEL
LIN {X 0,Y 573.326,Z 127.067,A -85,B 0,C 180,E1 -2160.703,E2 -2160.703} C_VEL
LIN {X 0,Y 573.289,Z 127.071,A -85,B 0,C 180,E1 -2162.811,E2 -2162.811} C_VEL
LIN {X 0,Y 573.281,Z 127.069,A -85,B 0,C 180,E1 -2165.629,E2 -2165.629} C_VEL
LIN {X 0,Y 573.249,Z 127.078,A -85,B 0,C 180,E1 -2168.461,E2 -2168.461} C_VEL
LIN {X 0,Y 573.276,Z 127.069,A -85,B 0,C 180,E1 -2171.312,E2 -2171.312} C_VEL
LIN {X 0,Y 573.267,Z 127.074,A -85,B 0,C 180,E1 -2174.417,E2 -2174.417} C_VEL
LIN {X 0,Y 573.18,Z 127.081,A -85,B 0,C 180,E1 -2177.114,E2 -2177.114} C_VEL
LIN {X 0,Y 573.268,Z 127.074,A -85,B 0,C 180,E1 -2179.33,E2 -2179.33} C_VEL
LIN {X 0,Y 573.198,Z 127.08,A -85,B 0,C 180,E1 -2182.34,E2 -2182.34} C_VEL
LIN {X 0,Y 573.23,Z 127.083,A -85,B 0,C 180,E1 -2185.412,E2 -2185.412} C_VEL
LIN {X 0,Y 573.196,Z 127.082,A -85,B 0,C 180,E1 -2188.018,E2 -2188.018} C_VEL
LIN {X 0,Y 573.203,Z 127.08,A -85,B 0,C 180,E1 -2190.877,E2 -2190.877} C_VEL
LIN {X 0,Y 573.218,Z 127.083,A -85,B 0,C 180,E1 -2193.517,E2 -2193.517} C_VEL
LIN {X 0,Y 573.177,Z 127.083,A -85,B 0,C 180,E1 -2196.055,E2 -2196.055} C_VEL
LIN {X 0,Y 573.176,Z 127.085,A -85,B 0,C 180,E1 -2198.707,E2 -2198.707} C_VEL
LIN {X 0,Y 573.192,Z 127.083,A -85,B 0,C 180,E1 -2201.588,E2 -2201.588} C_VEL
LIN {X 0,Y 573.21,Z 127.084,A -85,B 0,C 180,E1 -2204.673,E2 -2204.673} C_VEL
LIN {X 0,Y 573.206,Z 127.08,A -85,B 0,C 180,E1 -2207.596,E2 -2207.596} C_VEL
LIN {X 0,Y 573.233,Z 127.083,A -85,B 0,C 180,E1 -2210.57,E2 -2210.57} C_VEL
LIN {X 0,Y 573.231,Z 127.078,A -85,B 0,C 180,E1 -2213.076,E2 -2213.076} C_VEL
LIN {X 0,Y 573.247,Z 127.074,A -85,B 0,C 180,E1 -2215.67,E2 -2215.67} C_VEL
LIN {X 0,Y 573.227,Z 127.082,A -85,B 0,C 180,E1 -2218.184,E2 -2218.184} C_VEL
LIN {X 0,Y 573.239,Z 127.081,A -85,B 0,C 180,E1 -2220.633,E2 -2220.633} C_VEL
LIN {X 0,Y 573.21,Z 127.08,A -85,B 0,C 180,E1 -2223.514,E2 -2223.514} C_VEL
LIN {X 0,Y 573.204,Z 127.089,A -85,B 0,C 180,E1 -2226.133,E2 -2226.133} C_VEL
LIN {X 0,Y 573.236,Z 127.153,A -85,B 0,C 180,E1 -2226.586,E2 -2226.586} C_VEL
LIN {X 0,Y 573.96,Z 132.009,A -85,B 0,C 180,E1 -2227.312,E2 -2227.312} C_VEL
LIN {X 0,Y 573.785,Z 153.135,A -85,B 0,C 180,E1 -2230.316,E2 -2230.316} C_VEL
LIN {X 0,Y 573.588,Z 172.297,A -85,B 0,C 180,E1 -2233.015,E2 -2233.015} C_VEL
LIN {X 0,Y 573.407,Z 193.481,A -85,B 0,C 180,E1 -2235.991,E2 -2235.991} C_VEL
LIN {X 0,Y 573.389,Z 194.613,A -85,B 0,C 180,E1 -2236.149,E2 -2236.149} C_VEL
LIN {X 0,Y 574.049,Z 200.513,A -85,B 0,C 180,E1 -2236.256,E2 -2236.256} C_VEL
LIN {X 0,Y 573.883,Z 302.95,A -85,B 0,C 180,E1 -2237.558,E2 -2237.558} C_VEL
LIN {X 0,Y 573.779,Z 316.22,A -85,B 0,C 180,E1 -2237.87,E2 -2237.87} C_VEL
LIN {X 0,Y 573.699,Z 328.379,A -85,B 0,C 180,E1 -2238.294,E2 -2238.294} C_VEL
LIN {X 0,Y 573.586,Z 340.671,A -85,B 0,C 180,E1 -2238.876,E2 -2238.876} C_VEL
LIN {X 0,Y 573.428,Z 352.199,A -85,B 0,C 180,E1 -2239.585,E2 -2239.585} C_VEL
LIN {X 0,Y 573.333,Z 362.604,A -85,B 0,C 180,E1 -2240.386,E2 -2240.386} C_VEL
LIN {X 0,Y 573.241,Z 371.114,A -85,B 0,C 180,E1 -2241.185,E2 -2241.185} C_VEL
LIN {X 0,Y 573.161,Z 378.961,A -85,B 0,C 180,E1 -2242.071,E2 -2242.071} C_VEL
LIN {X 0,Y 573.073,Z 386.956,A -85,B 0,C 180,E1 -2243.186,E2 -2243.186} C_VEL
LIN {X 0,Y 573.07,Z 393.68,A -85,B 0,C 180,E1 -2244.37,E2 -2244.37} C_VEL
LIN {X 0,Y 573.028,Z 398.373,A -85,B 0,C 180,E1 -2245.428,E2 -2245.428} C_VEL
LIN {X 0,Y 573.022,Z 401.958,A -85,B 0,C 180,E1 -2246.484,E2 -2246.484} C_VEL
LIN {X 0,Y 572.959,Z 403.808,A -85,B 0,C 180,E1 -2247.188,E2 -2247.188} C_VEL
LIN {X 0,Y 572.946,Z 406.185,A -85,B 0,C 180,E1 -2248.594,E2 -2248.594} C_VEL
LIN {X 0,Y 572.938,Z 407,A -85,B 0,C 180,E1 -2250,E2 -2250} C_VEL
LIN {X 0,Y 572.946,Z 406.186,A -85,B 0,C 180,E1 -2251.406,E2 -2251.406} C_VEL
LIN {X 0,Y 572.94,Z 405.198,A -85,B 0,C 180,E1 -2252.109,E2 -2252.109} C_VEL
LIN {X 0,Y 572.959,Z 403.81,A -85,B 0,C 180,E1 -2252.812,E2 -2252.812} C_VEL
LIN {X 0,Y 573.015,Z 400.895,A -85,B 0,C 180,E1 -2253.868,E2 -2253.868} C_VEL
LIN {X 0,Y 572.963,Z 396.948,A -85,B 0,C 180,E1 -2254.926,E2 -2254.926} C_VEL
LIN {X 0,Y 573.065,Z 390.875,A -85,B 0,C 180,E1 -2256.16,E2 -2256.16} C_VEL
LIN {X 0,Y 573.12,Z 384.235,A -85,B 0,C 180,E1 -2257.221,E2 -2257.221} C_VEL
LIN {X 0,Y 573.201,Z 375.989,A -85,B 0,C 180,E1 -2258.283,E2 -2258.283} C_VEL
